SPLINE
SPL {X  -159.063, Y  +688.696, Z    +0.000, E1   +17.094, E3 -430810.553}
SPL {X  -159.987, Y  +672.488, Z    +0.000, E1    +5.638, E3 -430834.618}
SPL {X  -159.990, Y  +663.928, Z    +0.000, E1    -0.338, E3 -430840.413}
SPL {X  -159.990, Y  +658.009, Z    +0.000, E1    -4.774, E3 -430844.113}
SPL {X  -159.990, Y  +651.567, Z    +0.000, E1    -9.674, E3 -430849.516}
SPL {X  -159.990, Y  +638.711, Z    +0.000, E1   -17.883, E3 -430865.162}
SPL {X  -159.990, Y  +631.642, Z    +0.000, E1   -20.884, E3 -430880.721}
SPL {X  -159.990, Y  +626.048, Z    +0.000, E1   -22.026, E3 -430900.714}
SPL {X  -159.990, Y  +623.760, Z    +0.000, E1   -22.031, E3 -430912.701}
SPL {X  -159.990, Y  +621.334, Z    +0.000, E1   -22.029, E3 -430925.427}
SPL {X  -159.990, Y  +618.387, Z    +0.000, E1   -22.057, E3 -430940.817}
SPL {X  -159.990, Y  +615.830, Z    +0.000, E1   -22.023, E3 -430954.309}
SPL {X  -159.990, Y  +614.007, Z    +0.000, E1   -22.018, E3 -430963.886}
SPL {X  -159.990, Y  +611.459, Z    +0.000, E1   -22.053, E3 -430977.173}
SPL {X  -159.990, Y  +608.810, Z    +0.000, E1   -22.023, E3 -430991.141}
SPL {X  -159.990, Y  +606.481, Z    +0.000, E1   -22.033, E3 -431003.316}
SPL {X  -159.990, Y  +603.419, Z    +0.000, E1   -22.064, E3 -431019.256}
SPL {X  -159.990, Y  +600.642, Z    +0.000, E1   -22.032, E3 -431033.885}
SPL {X  -159.990, Y  +598.568, Z    +0.000, E1   -22.046, E3 -431044.678}
SPL {X  -159.990, Y  +595.493, Z    +0.000, E1   -22.070, E3 -431060.761}
SPL {X  -159.990, Y  +592.865, Z    +0.000, E1   -22.036, E3 -431074.590}
SPL {X  -159.990, Y  +590.803, Z    +0.000, E1   -22.046, E3 -431085.381}
SPL {X  -159.990, Y  +587.778, Z    +0.000, E1   -22.073, E3 -431101.156}
SPL {X  -159.990, Y  +585.120, Z    +0.000, E1   -22.045, E3 -431115.100}
SPL {X  -159.990, Y  +583.118, Z    +0.000, E1   -22.052, E3 -431125.586}
SPL {X  -159.990, Y  +580.862, Z    +0.000, E1   -22.049, E3 -431137.424}
SPL {X  -159.990, Y  +578.386, Z    +0.000, E1   -22.057, E3 -431150.379}
SPL {X  -159.990, Y  +576.252, Z    +0.000, E1   -22.038, E3 -431161.602}
SPL {X  -159.990, Y  +574.280, Z    +0.000, E1   -22.051, E3 -431171.896}
SPL {X  -159.990, Y  +571.711, Z    +0.000, E1   -22.058, E3 -431185.370}
SPL {X  -159.990, Y  +569.285, Z    +0.000, E1   -22.044, E3 -431198.095}
SPL {X  -159.990, Y  +567.211, Z    +0.000, E1   -22.046, E3 -431208.956}
SPL {X  -159.990, Y  +565.039, Z    +0.000, E1   -22.047, E3 -431220.334}
SPL {X  -159.990, Y  +562.755, Z    +0.000, E1   -22.047, E3 -431232.319}
SPL {X  -159.990, Y  +560.652, Z    +0.000, E1   -22.038, E3 -431243.364}
SPL {X  -159.990, Y  +558.852, Z    +0.000, E1   -22.046, E3 -431252.736}
SPL {X  -159.990, Y  +556.672, Z    +0.000, E1   -22.055, E3 -431264.126}
SPL {X  -159.990, Y  +553.726, Z    +0.000, E1   -22.080, E3 -431279.488}
SPL {X  -159.990, Y  +550.886, Z    +0.000, E1   -22.056, E3 -431294.427}
SPL {X  -159.990, Y  +547.986, Z    +0.000, E1   -22.078, E3 -431309.546}
SPL {X  -159.990, Y  +545.350, Z    +0.000, E1   -22.053, E3 -431323.407}
SPL {X  -159.990, Y  +543.405, Z    +0.000, E1   -22.048, E3 -431333.620}
SPL {X  -159.990, Y  +541.673, Z    +0.000, E1   -22.053, E3 -431342.684}
SPL {X  -159.990, Y  +539.341, Z    +0.000, E1   -22.056, E3 -431354.889}
SPL {X  -159.990, Y  +536.984, Z    +0.000, E1   -22.057, E3 -431367.221}
SPL {X  -159.990, Y  +534.045, Z    +0.000, E1   -22.087, E3 -431382.545}
SPL {X  -159.990, Y  +530.476, Z    +0.000, E1   -22.084, E3 -431401.239}
SPL {X  -159.990, Y  +527.412, Z    +0.000, E1   -22.067, E3 -431417.302}
SPL {X  -159.990, Y  +524.425, Z    +0.000, E1   -22.078, E3 -431432.935}
SPL {X  -159.990, Y  +521.599, Z    +0.000, E1   -22.060, E3 -431447.777}
SPL {X  -159.990, Y  +519.209, Z    +0.000, E1   -22.063, E3 -431460.252}
SPL {X  -159.990, Y  +516.651, Z    +0.000, E1   -22.071, E3 -431473.631}
SPL {X  -159.990, Y  +514.122, Z    +0.000, E1   -22.061, E3 -431486.903}
SPL {X  -159.990, Y  +511.670, Z    +0.000, E1   -22.064, E3 -431499.753}
SPL {X  -159.990, Y  +506.947, Z    +0.000, E1   -23.726, E3 -431509.781}
SPL {X  -159.990, Y  +496.921, Z    +0.000, E1   -28.340, E3 -431518.530}
SPL {X  -159.990, Y  +495.822, Z    +0.000, E1   -27.449, E3 -431529.278}
SPL {X  -159.990, Y  +494.952, Z    +0.000, E1   -26.628, E3 -431538.861}
SPL {X  -159.990, Y  +493.896, Z    +0.000, E1   -25.736, E3 -431550.191}
SPL {X  -159.990, Y  +491.647, Z    +0.000, E1   -25.401, E3 -431562.726}
SPL {X  -159.990, Y  +488.807, Z    +0.000, E1   -25.397, E3 -431575.425}
SPL {X  -159.990, Y  +486.070, Z    +0.000, E1   -25.399, E3 -431587.656}
SPL {X  -159.990, Y  +483.747, Z    +0.000, E1   -25.384, E3 -431598.069}
SPL {X  -159.990, Y  +481.038, Z    +0.000, E1   -25.412, E3 -431610.124}
SPL {X  -159.990, Y  +477.508, Z    +0.000, E1   -25.410, E3 -431625.906}
SPL {X  -159.990, Y  +473.634, Z    +0.000, E1   -25.426, E3 -431643.195}
SPL {X  -159.990, Y  +470.047, Z    +0.000, E1   -25.402, E3 -431659.276}
SPL {X  -159.990, Y  +467.082, Z    +0.000, E1   -25.399, E3 -431672.523}
SPL {X  -159.990, Y  +464.063, Z    +0.000, E1   -25.405, E3 -431686.018}
SPL {X  -159.990, Y  +460.712, Z    +0.000, E1   -25.411, E3 -431700.978}
SPL {X  -159.990, Y  +457.497, Z    +0.000, E1   -25.403, E3 -431715.350}
SPL {X  -159.990, Y  +455.126, Z    +0.000, E1   -25.389, E3 -431725.959}
SPL {X  -159.990, Y  +452.123, Z    +0.000, E1   -25.426, E3 -431739.317}
SPL {X  -159.990, Y  +448.503, Z    +0.000, E1   -25.410, E3 -431755.518}
SPL {X  -159.990, Y  +445.108, Z    +0.000, E1   -25.407, E3 -431770.756}
SPL {X  -159.990, Y  +441.797, Z    +0.000, E1   -25.390, E3 -431785.635}
SPL {X  -159.990, Y  +439.442, Z    +0.000, E1   -25.369, E3 -431796.212}
SPL {X  -159.990, Y  +436.316, Z    +0.000, E1   -25.420, E3 -431810.094}
SPL {X  -159.990, Y  +432.613, Z    +0.000, E1   -25.390, E3 -431826.719}
SPL {X  -159.990, Y  +429.079, Z    +0.000, E1   -25.407, E3 -431842.490}
SPL {X  -159.990, Y  +425.142, Z    +0.000, E1   -25.407, E3 -431860.092}
SPL {X  -159.990, Y  +421.010, Z    +0.000, E1   -25.418, E3 -431878.554}
SPL {X  -159.990, Y  +417.514, Z    +0.000, E1   -25.386, E3 -431894.246}
SPL {X  -159.990, Y  +414.805, Z    +0.000, E1   -25.385, E3 -431906.367}
SPL {X  -159.990, Y  +411.959, Z    +0.000, E1   -25.386, E3 -431919.093}
SPL {X  -159.990, Y  +408.981, Z    +0.000, E1   -25.392, E3 -431932.397}
SPL {X  -159.990, Y  +405.773, Z    +0.000, E1   -25.398, E3 -431946.707}
SPL {X  -159.990, Y  +402.805, Z    +0.000, E1   -25.389, E3 -431959.993}
SPL {X  -159.990, Y  +400.083, Z    +0.000, E1   -25.388, E3 -431972.170}
SPL {X  -159.990, Y  +396.740, Z    +0.000, E1   -25.410, E3 -431987.094}
SPL {X  -159.990, Y  +392.622, Z    +0.000, E1   -25.413, E3 -432005.522}
SPL {X  -159.990, Y  +388.328, Z    +0.000, E1   -25.413, E3 -432024.750}
SPL {X  -159.990, Y  +384.900, Z    +0.000, E1   -25.383, E3 -432040.112}
SPL {X  -159.990, Y  +382.110, Z    +0.000, E1   -25.393, E3 -432052.559}
SPL {X  -159.961, Y  +379.439, Z    +0.000, E1   -25.380, E3 -432064.538}
SPL {X  -159.894, Y  +376.959, Z    +0.000, E1   -25.370, E3 -432075.715}
SPL {X  -159.784, Y  +374.382, Z    +0.000, E1   -25.356, E3 -432087.356}
SPL {X  -159.621, Y  +371.640, Z    +0.000, E1   -25.335, E3 -432099.796}
SPL {X  -159.406, Y  +368.844, Z    +0.000, E1   -25.307, E3 -432112.509}
SPL {X  -159.144, Y  +366.072, Z    +0.000, E1   -25.281, E3 -432125.117}
SPL {X  -158.822, Y  +363.200, Z    +0.000, E1   -25.236, E3 -432138.289}
SPL {X  -158.491, Y  +360.654, Z    +0.000, E1   -25.188, E3 -432150.029}
SPL {X  -158.127, Y  +358.155, Z    +0.000, E1   -25.126, E3 -432161.649}
SPL {X  -158.095, Y  +357.947, Z    +0.000, E1   -21.741, E3 -432193.221}
ENDSPLINE

SPLINE
SPL {X  -158.454, Y  +360.384, Z    +0.000, E1   -19.366, E3 -432205.372}
SPL {X  -159.737, Y  +373.507, Z    +0.000, E1   -10.311, E3 -432227.408}
SPL {X  -159.990, Y  +382.574, Z    +0.000, E1    -4.463, E3 -432234.095}
SPL {X  -159.990, Y  +387.496, Z    +0.000, E1    -1.004, E3 -432236.841}
SPL {X  -159.990, Y  +395.121, Z    +0.000, E1    +4.514, E3 -432241.153}
SPL {X  -159.990, Y  +407.941, Z    +0.000, E1   +14.126, E3 -432253.227}
SPL {X  -159.990, Y  +418.671, Z    +0.000, E1   +19.855, E3 -432272.643}
SPL {X  -159.990, Y  +429.878, Z    +0.000, E1   +23.330, E3 -432302.698}
SPL {X  -159.990, Y  +432.766, Z    +0.000, E1   +23.321, E3 -432316.921}
SPL {X  -159.990, Y  +435.585, Z    +0.000, E1   +23.327, E3 -432330.801}
SPL {X  -159.990, Y  +439.169, Z    +0.000, E1   +23.353, E3 -432348.383}
SPL {X  -159.990, Y  +442.945, Z    +0.000, E1   +23.339, E3 -432367.001}
SPL {X  -159.990, Y  +446.037, Z    +0.000, E1   +23.324, E3 -432382.251}
SPL {X  -159.990, Y  +448.797, Z    +0.000, E1   +23.331, E3 -432395.781}
SPL {X  -159.990, Y  +451.747, Z    +0.000, E1   +23.333, E3 -432410.329}
SPL {X  -159.990, Y  +455.185, Z    +0.000, E1   +23.350, E3 -432427.189}
SPL {X  -159.990, Y  +458.265, Z    +0.000, E1   +23.328, E3 -432442.376}
SPL {X  -159.990, Y  +460.492, Z    +0.000, E1   +23.317, E3 -432453.375}
SPL {X  -159.990, Y  +462.929, Z    +0.000, E1   +23.331, E3 -432465.331}
SPL {X  -159.990, Y  +466.197, Z    +0.000, E1   +23.351, E3 -432481.368}
SPL {X  -159.990, Y  +468.951, Z    +0.000, E1   +23.319, E3 -432494.986}
SPL {X  -159.990, Y  +470.991, Z    +0.000, E1   +23.322, E3 -432505.015}
SPL {X  -159.990, Y  +474.027, Z    +0.000, E1   +23.352, E3 -432519.919}
SPL {X  -159.990, Y  +477.600, Z    +0.000, E1   +23.351, E3 -432537.523}
SPL {X  -159.990, Y  +481.169, Z    +0.000, E1   +23.337, E3 -432555.120}
SPL {X  -159.990, Y  +483.782, Z    +0.000, E1   +23.316, E3 -432568.025}
SPL {X  -159.990, Y  +486.109, Z    +0.000, E1   +23.322, E3 -432579.477}
SPL {X  -159.990, Y  +489.247, Z    +0.000, E1   +23.348, E3 -432594.864}
SPL {X  -159.990, Y  +493.031, Z    +0.000, E1   +23.350, E3 -432613.488}
SPL {X  -159.990, Y  +496.869, Z    +0.000, E1   +23.349, E3 -432632.379}
SPL {X  -159.990, Y  +499.995, Z    +0.000, E1   +23.324, E3 -432647.812}
SPL {X  -159.990, Y  +502.456, Z    +0.000, E1   +23.324, E3 -432659.927}
SPL {X  -159.990, Y  +504.508, Z    +0.000, E1   +23.311, E3 -432670.061}
SPL {X  -159.990, Y  +506.420, Z    +0.000, E1   +23.317, E3 -432679.453}
SPL {X  -159.990, Y  +508.862, Z    +0.000, E1   +23.328, E3 -432691.446}
SPL {X  -159.990, Y  +511.771, Z    +0.000, E1   +23.331, E3 -432705.768}
SPL {X  -159.990, Y  +514.757, Z    +0.000, E1   +23.329, E3 -432720.476}
SPL {X  -159.990, Y  +517.536, Z    +0.000, E1   +23.326, E3 -432734.142}
SPL {X  -159.990, Y  +519.961, Z    +0.000, E1   +23.334, E3 -432745.995}
SPL {X  -159.990, Y  +521.849, Z    +0.000, E1   +23.320, E3 -432755.317}
SPL {X  -159.990, Y  +523.968, Z    +0.000, E1   +23.332, E3 -432765.753}
SPL {X  -159.990, Y  +526.466, Z    +0.000, E1   +23.320, E3 -432778.096}
SPL {X  -159.990, Y  +528.815, Z    +0.000, E1   +23.322, E3 -432789.656}
SPL {X  -159.990, Y  +531.246, Z    +0.000, E1   +23.325, E3 -432801.594}
SPL {X  -159.990, Y  +534.143, Z    +0.000, E1   +23.341, E3 -432815.829}
SPL {X  -159.990, Y  +537.024, Z    +0.000, E1   +23.321, E3 -432830.073}
SPL {X  -159.990, Y  +539.129, Z    +0.000, E1   +23.310, E3 -432840.456}
SPL {X  -159.990, Y  +541.183, Z    +0.000, E1   +23.319, E3 -432850.553}
SPL {X  -159.990, Y  +544.314, Z    +0.000, E1   +23.352, E3 -432865.881}
SPL {X  -159.990, Y  +548.126, Z    +0.000, E1   +23.354, E3 -432884.636}
SPL {X  -159.990, Y  +551.344, Z    +0.000, E1   +23.327, E3 -432900.528}
SPL {X  -159.990, Y  +553.642, Z    +0.000, E1   +23.319, E3 -432911.847}
SPL {X  -159.990, Y  +556.481, Z    +0.000, E1   +23.354, E3 -432925.754}
SPL {X  -159.990, Y  +559.475, Z    +0.000, E1   +23.321, E3 -432940.559}
SPL {X  -159.990, Y  +561.830, Z    +0.000, E1   +23.325, E3 -432952.144}
SPL {X  -159.990, Y  +564.273, Z    +0.000, E1   +23.325, E3 -432964.168}
SPL {X  -159.990, Y  +567.351, Z    +0.000, E1   +23.348, E3 -432979.264}
SPL {X  -159.990, Y  +570.560, Z    +0.000, E1   +23.333, E3 -432995.093}
SPL {X  -159.990, Y  +572.975, Z    +0.000, E1   +23.316, E3 -433007.013}
SPL {X  -159.990, Y  +575.097, Z    +0.000, E1   +23.325, E3 -433017.440}
SPL {X  -159.990, Y  +577.540, Z    +0.000, E1   +23.325, E3 -433029.468}
SPL {X  -159.990, Y  +580.312, Z    +0.000, E1   +23.340, E3 -433043.050}
SPL {X  -159.990, Y  +583.018, Z    +0.000, E1   +23.331, E3 -433056.355}
SPL {X  -159.990, Y  +585.165, Z    +0.000, E1   +23.322, E3 -433066.971}
SPL {X  -159.990, Y  +587.388, Z    +0.000, E1   +23.328, E3 -433077.883}
SPL {X  -159.990, Y  +589.763, Z    +0.000, E1   +23.328, E3 -433089.570}
SPL {X  -159.990, Y  +592.397, Z    +0.000, E1   +23.344, E3 -433102.451}
SPL {X  -159.990, Y  +595.589, Z    +0.000, E1   +23.356, E3 -433118.124}
SPL {X  -159.990, Y  +598.571, Z    +0.000, E1   +23.347, E3 -433132.767}
SPL {X  -159.990, Y  +600.935, Z    +0.000, E1   +23.343, E3 -433144.360}
SPL {X  -159.990, Y  +603.047, Z    +0.000, E1   +23.344, E3 -433154.746}
SPL {X  -159.990, Y  +605.187, Z    +0.000, E1   +23.344, E3 -433165.268}
SPL {X  -159.990, Y  +607.319, Z    +0.000, E1   +23.353, E3 -433175.730}
SPL {X  -159.990, Y  +609.514, Z    +0.000, E1   +23.337, E3 -433186.560}
SPL {X  -159.990, Y  +611.376, Z    +0.000, E1   +23.336, E3 -433195.747}
SPL {X  -159.990, Y  +613.591, Z    +0.000, E1   +23.342, E3 -433206.624}
SPL {X  -159.990, Y  +615.604, Z    +0.000, E1   +23.330, E3 -433216.562}
SPL {X  -159.990, Y  +617.623, Z    +0.000, E1   +23.337, E3 -433226.492}
SPL {X  -159.990, Y  +620.788, Z    +0.000, E1   +23.368, E3 -433241.997}
SPL {X  -159.990, Y  +623.764, Z    +0.000, E1   +23.335, E3 -433256.690}
SPL {X  -159.990, Y  +625.941, Z    +0.000, E1   +23.337, E3 -433267.381}
SPL {X  -159.990, Y  +628.611, Z    +0.000, E1   +23.357, E3 -433280.460}
SPL {X  -159.990, Y  +631.169, Z    +0.000, E1   +23.338, E3 -433293.064}
SPL {X  -159.990, Y  +633.318, Z    +0.000, E1   +23.339, E3 -433303.653}
SPL {X  -159.990, Y  +635.650, Z    +0.000, E1   +23.339, E3 -433315.124}
SPL {X  -159.990, Y  +637.839, Z    +0.000, E1   +23.335, E3 -433325.934}
SPL {X  -159.990, Y  +640.072, Z    +0.000, E1   +23.325, E3 -433336.966}
SPL {X  -159.990, Y  +642.230, Z    +0.000, E1   +23.323, E3 -433347.648}
SPL {X  -159.990, Y  +645.287, Z    +0.000, E1   +23.340, E3 -433362.674}
SPL {X  -159.990, Y  +648.792, Z    +0.000, E1   +23.346, E3 -433379.933}
SPL {X  -159.990, Y  +652.623, Z    +0.000, E1   +23.348, E3 -433398.768}
SPL {X  -159.990, Y  +656.380, Z    +0.000, E1   +23.347, E3 -433417.262}
SPL {X  -159.990, Y  +659.180, Z    +0.000, E1   +23.314, E3 -433431.110}
SPL {X  -159.990, Y  +661.392, Z    +0.000, E1   +23.318, E3 -433442.004}
SPL {X  -159.990, Y  +663.662, Z    +0.000, E1   +23.322, E3 -433453.128}
SPL {X  -159.990, Y  +665.964, Z    +0.000, E1   +23.328, E3 -433464.419}
SPL {X  -159.990, Y  +668.989, Z    +0.000, E1   +23.359, E3 -433479.254}
SPL {X  -159.990, Y  +671.893, Z    +0.000, E1   +23.319, E3 -433493.634}
SPL {X  -159.974, Y  +673.789, Z    +0.000, E1   +23.323, E3 -433502.950}
SPL {X  -159.924, Y  +676.110, Z    +0.000, E1   +23.320, E3 -433514.435}
SPL {X  -159.801, Y  +679.265, Z    +0.000, E1   +23.327, E3 -433530.053}
SPL {X  -159.626, Y  +682.287, Z    +0.000, E1   +23.280, E3 -433545.152}
SPL {X  -159.462, Y  +684.486, Z    +0.000, E1   +23.258, E3 -433556.152}
SPL {X  -159.246, Y  +686.911, Z    +0.000, E1   +23.230, E3 -433568.313}
SPL {X  -159.019, Y  +689.098, Z    +0.000, E1   +23.200, E3 -433579.315}
SPL {X  -158.771, Y  +691.210, Z    +0.000, E1   +23.159, E3 -433589.990}
SPL {X  -158.553, Y  +692.896, Z    +0.000, E1   +23.130, E3 -433598.519}
ENDSPLINE

SPLINE
SPL {X  -159.063, Y  +688.696, Z    +0.000, E1   +17.094, E3 -433636.640}
SPL {X  -159.987, Y  +672.488, Z    +0.000, E1    +5.638, E3 -433660.705}
SPL {X  -159.990, Y  +663.928, Z    +0.000, E1    -0.338, E3 -433666.500}
SPL {X  -159.990, Y  +658.009, Z    +0.000, E1    -4.774, E3 -433670.200}
SPL {X  -159.990, Y  +651.567, Z    +0.000, E1    -9.674, E3 -433675.603}
SPL {X  -159.990, Y  +638.711, Z    +0.000, E1   -17.883, E3 -433691.249}
SPL {X  -159.990, Y  +631.642, Z    +0.000, E1   -20.884, E3 -433706.808}
SPL {X  -159.990, Y  +626.048, Z    +0.000, E1   -22.026, E3 -433726.801}
SPL {X  -159.990, Y  +623.760, Z    +0.000, E1   -22.031, E3 -433738.788}
SPL {X  -159.990, Y  +621.334, Z    +0.000, E1   -22.029, E3 -433751.514}
SPL {X  -159.990, Y  +619.505, Z    +0.000, E1   -22.018, E3 -433761.130}
SPL {X  -159.990, Y  +617.621, Z    +0.000, E1   -22.025, E3 -433770.996}
SPL {X  -159.990, Y  +615.830, Z    +0.000, E1   -22.023, E3 -433780.396}
SPL {X  -159.990, Y  +613.034, Z    +0.000, E1   -22.053, E3 -433795.002}
SPL {X  -159.990, Y  +609.503, Z    +0.000, E1   -22.054, E3 -433813.529}
SPL {X  -159.990, Y  +605.804, Z    +0.000, E1   -22.064, E3 -433832.873}
SPL {X  -159.990, Y  +602.819, Z    +0.000, E1   -22.037, E3 -433848.544}
SPL {X  -159.990, Y  +600.642, Z    +0.000, E1   -22.032, E3 -433859.972}
SPL {X  -159.990, Y  +598.568, Z    +0.000, E1   -22.046, E3 -433870.765}
SPL {X  -159.990, Y  +596.440, Z    +0.000, E1   -22.036, E3 -433881.947}
SPL {X  -159.990, Y  +593.768, Z    +0.000, E1   -22.071, E3 -433895.880}
SPL {X  -159.990, Y  +590.068, Z    +0.000, E1   -22.076, E3 -433915.248}
SPL {X  -159.990, Y  +587.130, Z    +0.000, E1   -22.046, E3 -433930.685}
SPL {X  -159.990, Y  +585.120, Z    +0.000, E1   -22.045, E3 -433941.187}
SPL {X  -159.990, Y  +583.118, Z    +0.000, E1   -22.052, E3 -433951.673}
SPL {X  -159.990, Y  +580.862, Z    +0.000, E1   -22.049, E3 -433963.511}
SPL {X  -159.990, Y  +578.386, Z    +0.000, E1   -22.057, E3 -433976.466}
SPL {X  -159.990, Y  +576.252, Z    +0.000, E1   -22.038, E3 -433987.689}
SPL {X  -159.990, Y  +574.280, Z    +0.000, E1   -22.051, E3 -433997.983}
SPL {X  -159.990, Y  +571.711, Z    +0.000, E1   -22.058, E3 -434011.457}
SPL {X  -159.990, Y  +569.285, Z    +0.000, E1   -22.044, E3 -434024.182}
SPL {X  -159.990, Y  +567.211, Z    +0.000, E1   -22.046, E3 -434035.043}
SPL {X  -159.990, Y  +565.039, Z    +0.000, E1   -22.047, E3 -434046.421}
SPL {X  -159.990, Y  +562.755, Z    +0.000, E1   -22.047, E3 -434058.406}
SPL {X  -159.990, Y  +559.661, Z    +0.000, E1   -22.078, E3 -434074.538}
SPL {X  -159.990, Y  +555.965, Z    +0.000, E1   -22.085, E3 -434093.847}
SPL {X  -159.990, Y  +553.115, Z    +0.000, E1   -22.054, E3 -434108.832}
SPL {X  -159.990, Y  +550.886, Z    +0.000, E1   -22.056, E3 -434120.514}
SPL {X  -159.990, Y  +547.986, Z    +0.000, E1   -22.078, E3 -434135.633}
SPL {X  -159.990, Y  +545.350, Z    +0.000, E1   -22.053, E3 -434149.494}
SPL {X  -159.990, Y  +543.405, Z    +0.000, E1   -22.048, E3 -434159.707}
SPL {X  -159.990, Y  +541.673, Z    +0.000, E1   -22.053, E3 -434168.771}
SPL {X  -159.990, Y  +539.341, Z    +0.000, E1   -22.056, E3 -434180.976}
SPL {X  -159.990, Y  +536.301, Z    +0.000, E1   -22.084, E3 -434196.831}
SPL {X  -159.990, Y  +533.389, Z    +0.000, E1   -22.057, E3 -434212.138}
SPL {X  -159.990, Y  +531.347, Z    +0.000, E1   -22.052, E3 -434222.839}
SPL {X  -159.990, Y  +528.972, Z    +0.000, E1   -22.072, E3 -434235.212}
SPL {X  -159.990, Y  +526.034, Z    +0.000, E1   -22.073, E3 -434250.591}
SPL {X  -159.990, Y  +523.717, Z    +0.000, E1   -22.050, E3 -434262.796}
SPL {X  -159.990, Y  +521.599, Z    +0.000, E1   -22.060, E3 -434273.864}
SPL {X  -159.990, Y  +519.209, Z    +0.000, E1   -22.063, E3 -434286.338}
SPL {X  -159.990, Y  +517.330, Z    +0.000, E1   -22.053, E3 -434296.194}
SPL {X  -159.990, Y  +514.729, Z    +0.000, E1   -22.089, E3 -434309.752}
SPL {X  -159.990, Y  +511.670, Z    +0.000, E1   -22.064, E3 -434325.840}
SPL {X  -159.990, Y  +506.947, Z    +0.000, E1   -23.726, E3 -434335.868}
SPL {X  -159.990, Y  +496.921, Z    +0.000, E1   -28.340, E3 -434344.617}
SPL {X  -159.990, Y  +495.822, Z    +0.000, E1   -27.449, E3 -434355.365}
SPL {X  -159.990, Y  +494.952, Z    +0.000, E1   -26.628, E3 -434364.948}
SPL {X  -159.990, Y  +493.896, Z    +0.000, E1   -25.736, E3 -434376.278}
SPL {X  -159.990, Y  +491.647, Z    +0.000, E1   -25.401, E3 -434388.813}
SPL {X  -159.990, Y  +488.807, Z    +0.000, E1   -25.397, E3 -434401.512}
SPL {X  -159.990, Y  +486.070, Z    +0.000, E1   -25.399, E3 -434413.743}
SPL {X  -159.990, Y  +482.821, Z    +0.000, E1   -25.411, E3 -434428.244}
SPL {X  -159.990, Y  +480.183, Z    +0.000, E1   -25.384, E3 -434440.084}
SPL {X  -159.990, Y  +477.508, Z    +0.000, E1   -25.410, E3 -434451.993}
SPL {X  -159.990, Y  +473.634, Z    +0.000, E1   -25.426, E3 -434469.282}
SPL {X  -159.990, Y  +470.047, Z    +0.000, E1   -25.402, E3 -434485.363}
SPL {X  -159.990, Y  +467.082, Z    +0.000, E1   -25.399, E3 -434498.610}
SPL {X  -159.990, Y  +464.063, Z    +0.000, E1   -25.405, E3 -434512.105}
SPL {X  -159.990, Y  +460.712, Z    +0.000, E1   -25.411, E3 -434527.065}
SPL {X  -159.990, Y  +457.497, Z    +0.000, E1   -25.403, E3 -434541.437}
SPL {X  -159.990, Y  +455.126, Z    +0.000, E1   -25.389, E3 -434552.046}
SPL {X  -159.990, Y  +453.438, Z    +0.000, E1   -25.385, E3 -434559.606}
SPL {X  -159.990, Y  +450.823, Z    +0.000, E1   -25.417, E3 -434571.225}
SPL {X  -159.990, Y  +446.894, Z    +0.000, E1   -25.428, E3 -434588.782}
SPL {X  -159.990, Y  +443.345, Z    +0.000, E1   -25.390, E3 -434604.790}
SPL {X  -159.990, Y  +441.077, Z    +0.000, E1   -25.369, E3 -434614.988}
SPL {X  -159.990, Y  +438.608, Z    +0.000, E1   -25.392, E3 -434625.985}
SPL {X  -159.990, Y  +434.852, Z    +0.000, E1   -25.415, E3 -434642.739}
SPL {X  -159.990, Y  +430.645, Z    +0.000, E1   -25.414, E3 -434661.559}
SPL {X  -159.990, Y  +426.865, Z    +0.000, E1   -25.398, E3 -434678.488}
SPL {X  -159.990, Y  +424.251, Z    +0.000, E1   -25.375, E3 -434690.225}
SPL {X  -159.990, Y  +421.010, Z    +0.000, E1   -25.418, E3 -434704.640}
SPL {X  -159.990, Y  +417.514, Z    +0.000, E1   -25.386, E3 -434720.333}
SPL {X  -159.990, Y  +414.805, Z    +0.000, E1   -25.385, E3 -434732.453}
SPL {X  -159.990, Y  +411.282, Z    +0.000, E1   -25.413, E3 -434748.154}
SPL {X  -159.990, Y  +408.351, Z    +0.000, E1   -25.372, E3 -434761.341}
SPL {X  -159.990, Y  +405.773, Z    +0.000, E1   -25.398, E3 -434772.794}
SPL {X  -159.990, Y  +402.805, Z    +0.000, E1   -25.389, E3 -434786.080}
SPL {X  -159.990, Y  +400.083, Z    +0.000, E1   -25.388, E3 -434798.257}
SPL {X  -159.990, Y  +396.740, Z    +0.000, E1   -25.410, E3 -434813.181}
SPL {X  -159.990, Y  +393.569, Z    +0.000, E1   -25.379, E3 -434827.431}
SPL {X  -159.990, Y  +390.564, Z    +0.000, E1   -25.393, E3 -434840.875}
SPL {X  -159.990, Y  +387.503, Z    +0.000, E1   -25.378, E3 -434854.589}
SPL {X  -159.990, Y  +384.900, Z    +0.000, E1   -25.383, E3 -434866.199}
SPL {X  -159.990, Y  +382.110, Z    +0.000, E1   -25.393, E3 -434878.646}
SPL {X  -159.961, Y  +379.439, Z    +0.000, E1   -25.380, E3 -434890.625}
SPL {X  -159.894, Y  +376.959, Z    +0.000, E1   -25.370, E3 -434901.802}
SPL {X  -159.784, Y  +374.382, Z    +0.000, E1   -25.356, E3 -434913.443}
SPL {X  -159.621, Y  +371.640, Z    +0.000, E1   -25.335, E3 -434925.883}
SPL {X  -159.406, Y  +368.844, Z    +0.000, E1   -25.307, E3 -434938.596}
SPL {X  -159.144, Y  +366.072, Z    +0.000, E1   -25.281, E3 -434951.204}
SPL {X  -158.822, Y  +363.200, Z    +0.000, E1   -25.236, E3 -434964.376}
SPL {X  -158.491, Y  +360.654, Z    +0.000, E1   -25.188, E3 -434976.116}
SPL {X  -158.127, Y  +358.155, Z    +0.000, E1   -25.126, E3 -434987.736}
SPL {X  -158.095, Y  +357.947, Z    +0.000, E1   -21.741, E3 -435019.308}
ENDSPLINE

SPLINE
SPL {X  -158.454, Y  +360.384, Z    +0.000, E1   -19.366, E3 -435031.459}
SPL {X  -159.737, Y  +373.507, Z    +0.000, E1   -10.311, E3 -435053.495}
SPL {X  -159.990, Y  +382.574, Z    +0.000, E1    -4.463, E3 -435060.182}
SPL {X  -159.990, Y  +389.909, Z    +0.000, E1    +0.662, E3 -435064.197}
SPL {X  -159.990, Y  +396.289, Z    +0.000, E1    +5.500, E3 -435067.977}
SPL {X  -159.990, Y  +407.941, Z    +0.000, E1   +14.126, E3 -435079.314}
SPL {X  -159.990, Y  +418.671, Z    +0.000, E1   +19.855, E3 -435098.730}
SPL {X  -159.990, Y  +429.878, Z    +0.000, E1   +23.330, E3 -435128.785}
SPL {X  -159.990, Y  +432.103, Z    +0.000, E1   +23.301, E3 -435139.804}
SPL {X  -159.990, Y  +434.188, Z    +0.000, E1   +23.325, E3 -435150.000}
SPL {X  -159.990, Y  +436.320, Z    +0.000, E1   +23.304, E3 -435160.553}
SPL {X  -159.990, Y  +439.169, Z    +0.000, E1   +23.353, E3 -435174.470}
SPL {X  -159.990, Y  +442.945, Z    +0.000, E1   +23.339, E3 -435193.088}
SPL {X  -159.990, Y  +446.037, Z    +0.000, E1   +23.324, E3 -435208.338}
SPL {X  -159.990, Y  +448.797, Z    +0.000, E1   +23.331, E3 -435221.868}
SPL {X  -159.990, Y  +451.747, Z    +0.000, E1   +23.333, E3 -435236.416}
SPL {X  -159.990, Y  +455.185, Z    +0.000, E1   +23.350, E3 -435253.276}
SPL {X  -159.990, Y  +458.265, Z    +0.000, E1   +23.328, E3 -435268.463}
SPL {X  -159.990, Y  +460.492, Z    +0.000, E1   +23.317, E3 -435279.462}
SPL {X  -159.990, Y  +462.929, Z    +0.000, E1   +23.331, E3 -435291.418}
SPL {X  -159.990, Y  +465.027, Z    +0.000, E1   +23.313, E3 -435301.771}
SPL {X  -159.990, Y  +466.881, Z    +0.000, E1   +23.322, E3 -435310.880}
SPL {X  -159.990, Y  +468.951, Z    +0.000, E1   +23.319, E3 -435321.072}
SPL {X  -159.990, Y  +471.818, Z    +0.000, E1   +23.351, E3 -435335.119}
SPL {X  -159.990, Y  +474.801, Z    +0.000, E1   +23.320, E3 -435349.895}
SPL {X  -159.990, Y  +476.830, Z    +0.000, E1   +23.323, E3 -435359.874}
SPL {X  -159.990, Y  +479.553, Z    +0.000, E1   +23.328, E3 -435373.276}
SPL {X  -159.990, Y  +481.893, Z    +0.000, E1   +23.312, E3 -435384.826}
SPL {X  -159.990, Y  +483.782, Z    +0.000, E1   +23.316, E3 -435394.112}
SPL {X  -159.990, Y  +486.109, Z    +0.000, E1   +23.322, E3 -435405.564}
SPL {X  -159.990, Y  +489.247, Z    +0.000, E1   +23.348, E3 -435420.951}
SPL {X  -159.990, Y  +493.031, Z    +0.000, E1   +23.350, E3 -435439.575}
SPL {X  -159.990, Y  +496.869, Z    +0.000, E1   +23.349, E3 -435458.466}
SPL {X  -159.990, Y  +499.995, Z    +0.000, E1   +23.324, E3 -435473.899}
SPL {X  -159.990, Y  +502.456, Z    +0.000, E1   +23.324, E3 -435486.014}
SPL {X  -159.990, Y  +505.646, Z    +0.000, E1   +23.350, E3 -435501.669}
SPL {X  -159.990, Y  +508.862, Z    +0.000, E1   +23.328, E3 -435517.533}
SPL {X  -159.990, Y  +511.771, Z    +0.000, E1   +23.331, E3 -435531.855}
SPL {X  -159.990, Y  +514.016, Z    +0.000, E1   +23.308, E3 -435542.959}
SPL {X  -159.990, Y  +516.860, Z    +0.000, E1   +23.355, E3 -435556.845}
SPL {X  -159.990, Y  +520.719, Z    +0.000, E1   +23.363, E3 -435575.755}
SPL {X  -159.990, Y  +523.968, Z    +0.000, E1   +23.332, E3 -435591.840}
SPL {X  -159.990, Y  +526.466, Z    +0.000, E1   +23.320, E3 -435604.183}
SPL {X  -159.990, Y  +528.815, Z    +0.000, E1   +23.322, E3 -435615.743}
SPL {X  -159.990, Y  +531.246, Z    +0.000, E1   +23.325, E3 -435627.681}
SPL {X  -159.990, Y  +533.354, Z    +0.000, E1   +23.318, E3 -435638.067}
SPL {X  -159.990, Y  +534.931, Z    +0.000, E1   +23.312, E3 -435645.861}
SPL {X  -159.990, Y  +537.024, Z    +0.000, E1   +23.321, E3 -435656.160}
SPL {X  -159.990, Y  +539.129, Z    +0.000, E1   +23.310, E3 -435666.543}
SPL {X  -159.990, Y  +541.183, Z    +0.000, E1   +23.319, E3 -435676.640}
SPL {X  -159.990, Y  +544.314, Z    +0.000, E1   +23.352, E3 -435691.968}
SPL {X  -159.990, Y  +548.126, Z    +0.000, E1   +23.354, E3 -435710.723}
SPL {X  -159.990, Y  +551.344, Z    +0.000, E1   +23.327, E3 -435726.615}
SPL {X  -159.990, Y  +553.642, Z    +0.000, E1   +23.319, E3 -435737.934}
SPL {X  -159.990, Y  +556.481, Z    +0.000, E1   +23.354, E3 -435751.841}
SPL {X  -159.990, Y  +559.475, Z    +0.000, E1   +23.321, E3 -435766.646}
SPL {X  -159.990, Y  +561.830, Z    +0.000, E1   +23.325, E3 -435778.231}
SPL {X  -159.990, Y  +564.273, Z    +0.000, E1   +23.325, E3 -435790.255}
SPL {X  -159.990, Y  +567.351, Z    +0.000, E1   +23.348, E3 -435805.351}
SPL {X  -159.990, Y  +570.560, Z    +0.000, E1   +23.333, E3 -435821.180}
SPL {X  -159.990, Y  +572.975, Z    +0.000, E1   +23.316, E3 -435833.100}
SPL {X  -159.990, Y  +575.097, Z    +0.000, E1   +23.325, E3 -435843.527}
SPL {X  -159.990, Y  +577.540, Z    +0.000, E1   +23.325, E3 -435855.555}
SPL {X  -159.990, Y  +580.312, Z    +0.000, E1   +23.340, E3 -435869.137}
SPL {X  -159.990, Y  +583.018, Z    +0.000, E1   +23.331, E3 -435882.442}
SPL {X  -159.990, Y  +585.165, Z    +0.000, E1   +23.322, E3 -435893.058}
SPL {X  -159.990, Y  +587.388, Z    +0.000, E1   +23.328, E3 -435903.970}
SPL {X  -159.990, Y  +589.763, Z    +0.000, E1   +23.328, E3 -435915.657}
SPL {X  -159.990, Y  +592.397, Z    +0.000, E1   +23.344, E3 -435928.538}
SPL {X  -159.990, Y  +595.589, Z    +0.000, E1   +23.356, E3 -435944.211}
SPL {X  -159.990, Y  +598.571, Z    +0.000, E1   +23.347, E3 -435958.854}
SPL {X  -159.990, Y  +600.935, Z    +0.000, E1   +23.343, E3 -435970.447}
SPL {X  -159.990, Y  +603.047, Z    +0.000, E1   +23.344, E3 -435980.833}
SPL {X  -159.990, Y  +605.187, Z    +0.000, E1   +23.344, E3 -435991.355}
SPL {X  -159.990, Y  +607.319, Z    +0.000, E1   +23.353, E3 -436001.817}
SPL {X  -159.990, Y  +609.514, Z    +0.000, E1   +23.337, E3 -436012.646}
SPL {X  -159.990, Y  +611.376, Z    +0.000, E1   +23.336, E3 -436021.834}
SPL {X  -159.990, Y  +613.591, Z    +0.000, E1   +23.342, E3 -436032.711}
SPL {X  -159.990, Y  +615.604, Z    +0.000, E1   +23.330, E3 -436042.649}
SPL {X  -159.990, Y  +617.623, Z    +0.000, E1   +23.337, E3 -436052.579}
SPL {X  -159.990, Y  +620.788, Z    +0.000, E1   +23.368, E3 -436068.084}
SPL {X  -159.990, Y  +623.764, Z    +0.000, E1   +23.335, E3 -436082.777}
SPL {X  -159.990, Y  +625.941, Z    +0.000, E1   +23.337, E3 -436093.468}
SPL {X  -159.990, Y  +628.611, Z    +0.000, E1   +23.357, E3 -436106.547}
SPL {X  -159.990, Y  +631.169, Z    +0.000, E1   +23.338, E3 -436119.151}
SPL {X  -159.990, Y  +633.318, Z    +0.000, E1   +23.339, E3 -436129.740}
SPL {X  -159.990, Y  +635.650, Z    +0.000, E1   +23.339, E3 -436141.211}
SPL {X  -159.990, Y  +637.839, Z    +0.000, E1   +23.335, E3 -436152.021}
SPL {X  -159.990, Y  +640.072, Z    +0.000, E1   +23.325, E3 -436163.053}
SPL {X  -159.990, Y  +642.230, Z    +0.000, E1   +23.323, E3 -436173.735}
SPL {X  -159.990, Y  +645.287, Z    +0.000, E1   +23.340, E3 -436188.761}
SPL {X  -159.990, Y  +648.792, Z    +0.000, E1   +23.346, E3 -436206.020}
SPL {X  -159.990, Y  +652.623, Z    +0.000, E1   +23.348, E3 -436224.854}
SPL {X  -159.990, Y  +656.380, Z    +0.000, E1   +23.347, E3 -436243.349}
SPL {X  -159.990, Y  +659.180, Z    +0.000, E1   +23.314, E3 -436257.197}
SPL {X  -159.990, Y  +661.392, Z    +0.000, E1   +23.318, E3 -436268.091}
SPL {X  -159.990, Y  +663.662, Z    +0.000, E1   +23.322, E3 -436279.215}
SPL {X  -159.990, Y  +665.964, Z    +0.000, E1   +23.328, E3 -436290.506}
SPL {X  -159.990, Y  +668.989, Z    +0.000, E1   +23.359, E3 -436305.341}
SPL {X  -159.983, Y  +672.946, Z    +0.000, E1   +23.359, E3 -436324.823}
SPL {X  -159.924, Y  +676.110, Z    +0.000, E1   +23.320, E3 -436340.522}
SPL {X  -159.801, Y  +679.265, Z    +0.000, E1   +23.327, E3 -436356.140}
SPL {X  -159.626, Y  +682.287, Z    +0.000, E1   +23.280, E3 -436371.239}
SPL {X  -159.462, Y  +684.486, Z    +0.000, E1   +23.258, E3 -436382.239}
SPL {X  -159.246, Y  +686.911, Z    +0.000, E1   +23.230, E3 -436394.400}
SPL {X  -159.019, Y  +689.098, Z    +0.000, E1   +23.200, E3 -436405.402}
SPL {X  -158.660, Y  +692.086, Z    +0.000, E1   +23.176, E3 -436420.446}
ENDSPLINE

SPLINE
SPL {X  -159.063, Y  +688.696, Z    +0.000, E1   +17.094, E3 -436462.727}
SPL {X  -159.967, Y  +674.206, Z    +0.000, E1    +6.731, E3 -436485.540}
SPL {X  -159.990, Y  +665.270, Z    +0.000, E1    +0.699, E3 -436491.710}
SPL {X  -159.990, Y  +658.009, Z    +0.000, E1    -4.774, E3 -436496.287}
SPL {X  -159.990, Y  +651.567, Z    +0.000, E1    -9.674, E3 -436501.690}
SPL {X  -159.990, Y  +637.762, Z    +0.000, E1   -18.345, E3 -436519.048}
SPL {X  -159.990, Y  +626.382, Z    +0.000, E1   -22.040, E3 -436551.097}
SPL {X  -159.990, Y  +623.760, Z    +0.000, E1   -22.031, E3 -436564.875}
SPL {X  -159.990, Y  +621.334, Z    +0.000, E1   -22.029, E3 -436577.601}
SPL {X  -159.990, Y  +619.505, Z    +0.000, E1   -22.018, E3 -436587.217}
SPL {X  -159.990, Y  +617.621, Z    +0.000, E1   -22.025, E3 -436597.083}
SPL {X  -159.990, Y  +614.928, Z    +0.000, E1   -22.055, E3 -436611.144}
SPL {X  -159.990, Y  +611.459, Z    +0.000, E1   -22.053, E3 -436629.347}
SPL {X  -159.990, Y  +608.810, Z    +0.000, E1   -22.023, E3 -436643.315}
SPL {X  -159.990, Y  +605.804, Z    +0.000, E1   -22.064, E3 -436658.960}
SPL {X  -159.990, Y  +602.819, Z    +0.000, E1   -22.037, E3 -436674.631}
SPL {X  -159.990, Y  +600.642, Z    +0.000, E1   -22.032, E3 -436686.059}
SPL {X  -159.990, Y  +598.568, Z    +0.000, E1   -22.046, E3 -436696.852}
SPL {X  -159.990, Y  +596.440, Z    +0.000, E1   -22.036, E3 -436708.034}
SPL {X  -159.990, Y  +593.768, Z    +0.000, E1   -22.071, E3 -436721.967}
SPL {X  -159.990, Y  +590.068, Z    +0.000, E1   -22.076, E3 -436741.335}
SPL {X  -159.990, Y  +587.130, Z    +0.000, E1   -22.046, E3 -436756.772}
SPL {X  -159.990, Y  +585.120, Z    +0.000, E1   -22.045, E3 -436767.274}
SPL {X  -159.990, Y  +583.118, Z    +0.000, E1   -22.052, E3 -436777.760}
SPL {X  -159.990, Y  +580.862, Z    +0.000, E1   -22.049, E3 -436789.598}
SPL {X  -159.990, Y  +578.386, Z    +0.000, E1   -22.057, E3 -436802.553}
SPL {X  -159.990, Y  +576.252, Z    +0.000, E1   -22.038, E3 -436813.776}
SPL {X  -159.990, Y  +574.280, Z    +0.000, E1   -22.051, E3 -436824.070}
SPL {X  -159.990, Y  +571.711, Z    +0.000, E1   -22.058, E3 -436837.544}
SPL {X  -159.990, Y  +569.285, Z    +0.000, E1   -22.044, E3 -436850.269}
SPL {X  -159.990, Y  +567.211, Z    +0.000, E1   -22.046, E3 -436861.130}
SPL {X  -159.990, Y  +565.039, Z    +0.000, E1   -22.047, E3 -436872.508}
SPL {X  -159.990, Y  +562.755, Z    +0.000, E1   -22.047, E3 -436884.493}
SPL {X  -159.990, Y  +560.652, Z    +0.000, E1   -22.038, E3 -436895.538}
SPL {X  -159.990, Y  +558.852, Z    +0.000, E1   -22.046, E3 -436904.910}
SPL {X  -159.990, Y  +556.672, Z    +0.000, E1   -22.055, E3 -436916.300}
SPL {X  -159.990, Y  +553.726, Z    +0.000, E1   -22.080, E3 -436931.662}
SPL {X  -159.990, Y  +550.886, Z    +0.000, E1   -22.056, E3 -436946.601}
SPL {X  -159.990, Y  +548.814, Z    +0.000, E1   -22.049, E3 -436957.447}
SPL {X  -159.990, Y  +546.122, Z    +0.000, E1   -22.088, E3 -436971.460}
SPL {X  -159.990, Y  +542.390, Z    +0.000, E1   -22.086, E3 -436991.042}
SPL {X  -159.990, Y  +539.341, Z    +0.000, E1   -22.056, E3 -437007.063}
SPL {X  -159.990, Y  +536.984, Z    +0.000, E1   -22.057, E3 -437019.395}
SPL {X  -159.990, Y  +534.045, Z    +0.000, E1   -22.087, E3 -437034.719}
SPL {X  -159.990, Y  +530.476, Z    +0.000, E1   -22.084, E3 -437053.412}
SPL {X  -159.990, Y  +527.412, Z    +0.000, E1   -22.067, E3 -437069.476}
SPL {X  -159.990, Y  +525.349, Z    +0.000, E1   -22.050, E3 -437080.317}
SPL {X  -159.990, Y  +523.717, Z    +0.000, E1   -22.050, E3 -437088.883}
SPL {X  -159.990, Y  +521.599, Z    +0.000, E1   -22.060, E3 -437099.951}
SPL {X  -159.990, Y  +519.209, Z    +0.000, E1   -22.063, E3 -437112.425}
SPL {X  -159.990, Y  +517.330, Z    +0.000, E1   -22.053, E3 -437122.281}
SPL {X  -159.990, Y  +514.729, Z    +0.000, E1   -22.089, E3 -437135.839}
SPL {X  -159.990, Y  +511.670, Z    +0.000, E1   -22.064, E3 -437151.927}
SPL {X  -159.990, Y  +506.947, Z    +0.000, E1   -23.726, E3 -437161.955}
SPL {X  -159.990, Y  +496.921, Z    +0.000, E1   -28.340, E3 -437170.704}
SPL {X  -159.990, Y  +495.822, Z    +0.000, E1   -27.449, E3 -437181.452}
SPL {X  -159.990, Y  +494.952, Z    +0.000, E1   -26.628, E3 -437191.035}
SPL {X  -159.990, Y  +493.896, Z    +0.000, E1   -25.736, E3 -437202.365}
SPL {X  -159.990, Y  +491.647, Z    +0.000, E1   -25.401, E3 -437214.900}
SPL {X  -159.990, Y  +488.807, Z    +0.000, E1   -25.397, E3 -437227.599}
SPL {X  -159.990, Y  +486.070, Z    +0.000, E1   -25.399, E3 -437239.830}
SPL {X  -159.990, Y  +482.821, Z    +0.000, E1   -25.411, E3 -437254.331}
SPL {X  -159.990, Y  +480.183, Z    +0.000, E1   -25.384, E3 -437266.171}
SPL {X  -159.990, Y  +477.508, Z    +0.000, E1   -25.410, E3 -437278.080}
SPL {X  -159.990, Y  +473.634, Z    +0.000, E1   -25.426, E3 -437295.369}
SPL {X  -159.990, Y  +470.047, Z    +0.000, E1   -25.402, E3 -437311.450}
SPL {X  -159.990, Y  +466.213, Z    +0.000, E1   -25.433, E3 -437328.530}
SPL {X  -159.990, Y  +462.520, Z    +0.000, E1   -25.400, E3 -437345.098}
SPL {X  -159.990, Y  +460.081, Z    +0.000, E1   -25.390, E3 -437356.000}
SPL {X  -159.990, Y  +457.497, Z    +0.000, E1   -25.403, E3 -437367.524}
SPL {X  -159.990, Y  +454.323, Z    +0.000, E1   -25.412, E3 -437381.684}
SPL {X  -159.990, Y  +451.400, Z    +0.000, E1   -25.397, E3 -437394.774}
SPL {X  -159.990, Y  +448.503, Z    +0.000, E1   -25.410, E3 -437407.692}
SPL {X  -159.990, Y  +445.108, Z    +0.000, E1   -25.407, E3 -437422.930}
SPL {X  -159.990, Y  +441.797, Z    +0.000, E1   -25.390, E3 -437437.809}
SPL {X  -159.990, Y  +439.442, Z    +0.000, E1   -25.369, E3 -437448.386}
SPL {X  -159.990, Y  +436.316, Z    +0.000, E1   -25.420, E3 -437462.268}
SPL {X  -159.990, Y  +432.613, Z    +0.000, E1   -25.390, E3 -437478.893}
SPL {X  -159.990, Y  +429.079, Z    +0.000, E1   -25.407, E3 -437494.664}
SPL {X  -159.990, Y  +426.149, Z    +0.000, E1   -25.374, E3 -437507.826}
SPL {X  -159.990, Y  +423.417, Z    +0.000, E1   -25.400, E3 -437519.991}
SPL {X  -159.990, Y  +420.283, Z    +0.000, E1   -25.386, E3 -437534.036}
SPL {X  -159.990, Y  +417.514, Z    +0.000, E1   -25.386, E3 -437546.420}
SPL {X  -159.990, Y  +414.805, Z    +0.000, E1   -25.385, E3 -437558.540}
SPL {X  -159.990, Y  +411.282, Z    +0.000, E1   -25.413, E3 -437574.241}
SPL {X  -159.990, Y  +407.450, Z    +0.000, E1   -25.401, E3 -437591.390}
SPL {X  -159.990, Y  +403.513, Z    +0.000, E1   -25.420, E3 -437608.944}
SPL {X  -159.990, Y  +399.257, Z    +0.000, E1   -25.420, E3 -437627.985}
SPL {X  -159.990, Y  +395.992, Z    +0.000, E1   -25.380, E3 -437642.674}
SPL {X  -159.990, Y  +393.569, Z    +0.000, E1   -25.379, E3 -437653.518}
SPL {X  -159.990, Y  +390.564, Z    +0.000, E1   -25.393, E3 -437666.962}
SPL {X  -159.990, Y  +387.503, Z    +0.000, E1   -25.378, E3 -437680.676}
SPL {X  -159.990, Y  +384.900, Z    +0.000, E1   -25.383, E3 -437692.286}
SPL {X  -159.990, Y  +382.110, Z    +0.000, E1   -25.393, E3 -437704.733}
SPL {X  -159.961, Y  +379.439, Z    +0.000, E1   -25.380, E3 -437716.712}
SPL {X  -159.894, Y  +376.959, Z    +0.000, E1   -25.370, E3 -437727.889}
SPL {X  -159.784, Y  +374.382, Z    +0.000, E1   -25.356, E3 -437739.530}
SPL {X  -159.621, Y  +371.640, Z    +0.000, E1   -25.335, E3 -437751.970}
SPL {X  -159.406, Y  +368.844, Z    +0.000, E1   -25.307, E3 -437764.683}
SPL {X  -159.144, Y  +366.072, Z    +0.000, E1   -25.281, E3 -437777.290}
SPL {X  -158.822, Y  +363.200, Z    +0.000, E1   -25.236, E3 -437790.463}
SPL {X  -158.491, Y  +360.654, Z    +0.000, E1   -25.188, E3 -437802.203}
SPL {X  -158.127, Y  +358.155, Z    +0.000, E1   -25.126, E3 -437813.823}
SPL {X  -158.095, Y  +357.947, Z    +0.000, E1   -21.741, E3 -437845.395}
ENDSPLINE

SPLINE
SPL {X  -158.454, Y  +360.384, Z    +0.000, E1   -19.366, E3 -437857.546}
SPL {X  -159.737, Y  +373.507, Z    +0.000, E1   -10.311, E3 -437879.582}
SPL {X  -159.990, Y  +382.574, Z    +0.000, E1    -4.463, E3 -437886.269}
SPL {X  -159.990, Y  +387.496, Z    +0.000, E1    -1.004, E3 -437889.014}
SPL {X  -159.990, Y  +395.121, Z    +0.000, E1    +4.514, E3 -437893.327}
SPL {X  -159.990, Y  +407.941, Z    +0.000, E1   +14.126, E3 -437905.401}
SPL {X  -159.990, Y  +418.671, Z    +0.000, E1   +19.855, E3 -437924.817}
SPL {X  -159.990, Y  +428.534, Z    +0.000, E1   +23.299, E3 -437948.337}
SPL {X  -159.990, Y  +430.313, Z    +0.000, E1   +23.313, E3 -437957.050}
SPL {X  -159.990, Y  +432.766, Z    +0.000, E1   +23.321, E3 -437969.095}
SPL {X  -159.990, Y  +434.794, Z    +0.000, E1   +23.304, E3 -437979.126}
SPL {X  -159.990, Y  +437.007, Z    +0.000, E1   +23.323, E3 -437989.978}
SPL {X  -159.990, Y  +439.778, Z    +0.000, E1   +23.323, E3 -438003.611}
SPL {X  -159.990, Y  +442.010, Z    +0.000, E1   +23.308, E3 -438014.632}
SPL {X  -159.990, Y  +443.729, Z    +0.000, E1   +23.310, E3 -438023.088}
SPL {X  -159.990, Y  +446.037, Z    +0.000, E1   +23.324, E3 -438034.425}
SPL {X  -159.990, Y  +449.434, Z    +0.000, E1   +23.356, E3 -438051.046}
SPL {X  -159.990, Y  +453.256, Z    +0.000, E1   +23.349, E3 -438069.881}
SPL {X  -159.990, Y  +455.953, Z    +0.000, E1   +23.320, E3 -438083.196}
SPL {X  -159.990, Y  +458.265, Z    +0.000, E1   +23.328, E3 -438094.550}
SPL {X  -159.990, Y  +461.258, Z    +0.000, E1   +23.344, E3 -438109.266}
SPL {X  -159.990, Y  +464.382, Z    +0.000, E1   +23.332, E3 -438124.647}
SPL {X  -159.990, Y  +466.881, Z    +0.000, E1   +23.322, E3 -438136.967}
SPL {X  -159.990, Y  +468.951, Z    +0.000, E1   +23.319, E3 -438147.159}
SPL {X  -159.990, Y  +470.991, Z    +0.000, E1   +23.322, E3 -438157.189}
SPL {X  -159.990, Y  +474.027, Z    +0.000, E1   +23.352, E3 -438172.093}
SPL {X  -159.990, Y  +477.600, Z    +0.000, E1   +23.351, E3 -438189.697}
SPL {X  -159.990, Y  +481.169, Z    +0.000, E1   +23.337, E3 -438207.294}
SPL {X  -159.990, Y  +483.782, Z    +0.000, E1   +23.316, E3 -438220.199}
SPL {X  -159.990, Y  +486.109, Z    +0.000, E1   +23.322, E3 -438231.651}
SPL {X  -159.990, Y  +489.247, Z    +0.000, E1   +23.348, E3 -438247.038}
SPL {X  -159.990, Y  +492.126, Z    +0.000, E1   +23.317, E3 -438261.273}
SPL {X  -159.990, Y  +494.937, Z    +0.000, E1   +23.343, E3 -438275.055}
SPL {X  -159.990, Y  +497.668, Z    +0.000, E1   +23.317, E3 -438288.548}
SPL {X  -159.990, Y  +499.995, Z    +0.000, E1   +23.324, E3 -438299.986}
SPL {X  -159.990, Y  +502.456, Z    +0.000, E1   +23.324, E3 -438312.100}
SPL {X  -159.990, Y  +504.508, Z    +0.000, E1   +23.311, E3 -438322.235}
SPL {X  -159.990, Y  +506.420, Z    +0.000, E1   +23.317, E3 -438331.627}
SPL {X  -159.990, Y  +508.862, Z    +0.000, E1   +23.328, E3 -438343.620}
SPL {X  -159.990, Y  +511.771, Z    +0.000, E1   +23.331, E3 -438357.942}
SPL {X  -159.990, Y  +514.757, Z    +0.000, E1   +23.329, E3 -438372.650}
SPL {X  -159.990, Y  +517.536, Z    +0.000, E1   +23.326, E3 -438386.316}
SPL {X  -159.990, Y  +519.961, Z    +0.000, E1   +23.334, E3 -438398.169}
SPL {X  -159.990, Y  +521.849, Z    +0.000, E1   +23.320, E3 -438407.491}
SPL {X  -159.990, Y  +523.968, Z    +0.000, E1   +23.332, E3 -438417.927}
SPL {X  -159.990, Y  +526.466, Z    +0.000, E1   +23.320, E3 -438430.270}
SPL {X  -159.990, Y  +528.815, Z    +0.000, E1   +23.322, E3 -438441.830}
SPL {X  -159.990, Y  +531.246, Z    +0.000, E1   +23.325, E3 -438453.768}
SPL {X  -159.990, Y  +533.354, Z    +0.000, E1   +23.318, E3 -438464.154}
SPL {X  -159.990, Y  +534.931, Z    +0.000, E1   +23.312, E3 -438471.948}
SPL {X  -159.990, Y  +537.024, Z    +0.000, E1   +23.321, E3 -438482.247}
SPL {X  -159.990, Y  +539.129, Z    +0.000, E1   +23.310, E3 -438492.630}
SPL {X  -159.990, Y  +541.183, Z    +0.000, E1   +23.319, E3 -438502.727}
SPL {X  -159.990, Y  +544.314, Z    +0.000, E1   +23.352, E3 -438518.055}
SPL {X  -159.990, Y  +548.126, Z    +0.000, E1   +23.354, E3 -438536.810}
SPL {X  -159.990, Y  +551.344, Z    +0.000, E1   +23.327, E3 -438552.702}
SPL {X  -159.990, Y  +553.642, Z    +0.000, E1   +23.319, E3 -438564.021}
SPL {X  -159.990, Y  +556.481, Z    +0.000, E1   +23.354, E3 -438577.928}
SPL {X  -159.990, Y  +559.475, Z    +0.000, E1   +23.321, E3 -438592.733}
SPL {X  -159.990, Y  +561.830, Z    +0.000, E1   +23.325, E3 -438604.318}
SPL {X  -159.990, Y  +564.273, Z    +0.000, E1   +23.325, E3 -438616.342}
SPL {X  -159.990, Y  +566.342, Z    +0.000, E1   +23.314, E3 -438626.547}
SPL {X  -159.990, Y  +568.849, Z    +0.000, E1   +23.338, E3 -438638.842}
SPL {X  -159.990, Y  +572.204, Z    +0.000, E1   +23.344, E3 -438655.337}
SPL {X  -159.990, Y  +575.097, Z    +0.000, E1   +23.325, E3 -438669.613}
SPL {X  -159.990, Y  +577.540, Z    +0.000, E1   +23.325, E3 -438681.642}
SPL {X  -159.990, Y  +580.312, Z    +0.000, E1   +23.340, E3 -438695.224}
SPL {X  -159.990, Y  +583.018, Z    +0.000, E1   +23.331, E3 -438708.529}
SPL {X  -159.990, Y  +585.165, Z    +0.000, E1   +23.322, E3 -438719.145}
SPL {X  -159.990, Y  +587.388, Z    +0.000, E1   +23.328, E3 -438730.057}
SPL {X  -159.990, Y  +589.763, Z    +0.000, E1   +23.328, E3 -438741.744}
SPL {X  -159.990, Y  +592.397, Z    +0.000, E1   +23.344, E3 -438754.625}
SPL {X  -159.990, Y  +594.928, Z    +0.000, E1   +23.334, E3 -438767.087}
SPL {X  -159.990, Y  +597.981, Z    +0.000, E1   +23.373, E3 -438782.002}
SPL {X  -159.990, Y  +600.935, Z    +0.000, E1   +23.343, E3 -438796.534}
SPL {X  -159.990, Y  +603.047, Z    +0.000, E1   +23.344, E3 -438806.920}
SPL {X  -159.990, Y  +605.187, Z    +0.000, E1   +23.344, E3 -438817.442}
SPL {X  -159.990, Y  +607.319, Z    +0.000, E1   +23.353, E3 -438827.904}
SPL {X  -159.990, Y  +610.569, Z    +0.000, E1   +23.372, E3 -438843.869}
SPL {X  -159.990, Y  +613.591, Z    +0.000, E1   +23.342, E3 -438858.798}
SPL {X  -159.990, Y  +615.604, Z    +0.000, E1   +23.330, E3 -438868.736}
SPL {X  -159.990, Y  +618.445, Z    +0.000, E1   +23.368, E3 -438882.649}
SPL {X  -159.990, Y  +621.517, Z    +0.000, E1   +23.337, E3 -438897.813}
SPL {X  -159.990, Y  +623.764, Z    +0.000, E1   +23.335, E3 -438908.863}
SPL {X  -159.990, Y  +625.941, Z    +0.000, E1   +23.337, E3 -438919.555}
SPL {X  -159.990, Y  +628.611, Z    +0.000, E1   +23.357, E3 -438932.634}
SPL {X  -159.990, Y  +631.169, Z    +0.000, E1   +23.338, E3 -438945.238}
SPL {X  -159.990, Y  +633.318, Z    +0.000, E1   +23.339, E3 -438955.827}
SPL {X  -159.990, Y  +635.650, Z    +0.000, E1   +23.339, E3 -438967.298}
SPL {X  -159.990, Y  +637.839, Z    +0.000, E1   +23.335, E3 -438978.108}
SPL {X  -159.990, Y  +640.072, Z    +0.000, E1   +23.325, E3 -438989.140}
SPL {X  -159.990, Y  +642.230, Z    +0.000, E1   +23.323, E3 -438999.822}
SPL {X  -159.990, Y  +645.287, Z    +0.000, E1   +23.340, E3 -439014.848}
SPL {X  -159.990, Y  +648.792, Z    +0.000, E1   +23.346, E3 -439032.107}
SPL {X  -159.990, Y  +651.647, Z    +0.000, E1   +23.312, E3 -439046.219}
SPL {X  -159.990, Y  +654.543, Z    +0.000, E1   +23.348, E3 -439060.385}
SPL {X  -159.990, Y  +658.319, Z    +0.000, E1   +23.349, E3 -439078.975}
SPL {X  -159.990, Y  +661.392, Z    +0.000, E1   +23.318, E3 -439094.178}
SPL {X  -159.990, Y  +663.662, Z    +0.000, E1   +23.322, E3 -439105.302}
SPL {X  -159.990, Y  +665.964, Z    +0.000, E1   +23.328, E3 -439116.592}
SPL {X  -159.990, Y  +667.870, Z    +0.000, E1   +23.320, E3 -439125.999}
SPL {X  -159.990, Y  +669.861, Z    +0.000, E1   +23.321, E3 -439135.800}
SPL {X  -159.983, Y  +672.946, Z    +0.000, E1   +23.359, E3 -439150.910}
SPL {X  -159.924, Y  +676.110, Z    +0.000, E1   +23.320, E3 -439166.609}
SPL {X  -159.845, Y  +678.302, Z    +0.000, E1   +23.298, E3 -439177.511}
SPL {X  -159.760, Y  +680.081, Z    +0.000, E1   +23.288, E3 -439186.354}
SPL {X  -159.626, Y  +682.287, Z    +0.000, E1   +23.280, E3 -439197.326}
SPL {X  -159.462, Y  +684.486, Z    +0.000, E1   +23.258, E3 -439208.325}
SPL {X  -159.246, Y  +686.911, Z    +0.000, E1   +23.230, E3 -439220.487}
SPL {X  -159.019, Y  +689.098, Z    +0.000, E1   +23.200, E3 -439231.489}
SPL {X  -158.771, Y  +691.210, Z    +0.000, E1   +23.159, E3 -439242.164}
SPL {X  -158.553, Y  +692.896, Z    +0.000, E1   +23.130, E3 -439250.693}
ENDSPLINE

SPLINE
SPL {X  -159.063, Y  +688.696, Z    +0.000, E1   +17.094, E3 -439288.814}
SPL {X  -159.987, Y  +672.488, Z    +0.000, E1    +5.638, E3 -439312.879}
SPL {X  -159.990, Y  +663.928, Z    +0.000, E1    -0.338, E3 -439318.674}
SPL {X  -159.990, Y  +658.009, Z    +0.000, E1    -4.774, E3 -439322.374}
SPL {X  -159.990, Y  +651.567, Z    +0.000, E1    -9.674, E3 -439327.777}
SPL {X  -159.990, Y  +637.762, Z    +0.000, E1   -18.345, E3 -439345.135}
SPL {X  -159.990, Y  +626.382, Z    +0.000, E1   -22.040, E3 -439377.184}
SPL {X  -159.990, Y  +623.760, Z    +0.000, E1   -22.031, E3 -439390.962}
SPL {X  -159.990, Y  +621.334, Z    +0.000, E1   -22.029, E3 -439403.688}
SPL {X  -159.990, Y  +618.387, Z    +0.000, E1   -22.057, E3 -439419.078}
SPL {X  -159.990, Y  +615.830, Z    +0.000, E1   -22.023, E3 -439432.569}
SPL {X  -159.990, Y  +613.034, Z    +0.000, E1   -22.053, E3 -439447.176}
SPL {X  -159.990, Y  +609.503, Z    +0.000, E1   -22.054, E3 -439465.703}
SPL {X  -159.990, Y  +605.804, Z    +0.000, E1   -22.064, E3 -439485.047}
SPL {X  -159.990, Y  +602.819, Z    +0.000, E1   -22.037, E3 -439500.718}
SPL {X  -159.990, Y  +600.642, Z    +0.000, E1   -22.032, E3 -439512.146}
SPL {X  -159.990, Y  +598.568, Z    +0.000, E1   -22.046, E3 -439522.939}
SPL {X  -159.990, Y  +595.493, Z    +0.000, E1   -22.070, E3 -439539.022}
SPL {X  -159.990, Y  +592.865, Z    +0.000, E1   -22.036, E3 -439552.851}
SPL {X  -159.990, Y  +590.803, Z    +0.000, E1   -22.046, E3 -439563.641}
SPL {X  -159.990, Y  +587.778, Z    +0.000, E1   -22.073, E3 -439579.417}
SPL {X  -159.990, Y  +585.120, Z    +0.000, E1   -22.045, E3 -439593.361}
SPL {X  -159.990, Y  +583.118, Z    +0.000, E1   -22.052, E3 -439603.847}
SPL {X  -159.990, Y  +580.131, Z    +0.000, E1   -22.078, E3 -439619.453}
SPL {X  -159.990, Y  +576.888, Z    +0.000, E1   -22.061, E3 -439636.483}
SPL {X  -159.990, Y  +574.280, Z    +0.000, E1   -22.051, E3 -439650.157}
SPL {X  -159.990, Y  +572.375, Z    +0.000, E1   -22.037, E3 -439660.196}
SPL {X  -159.990, Y  +569.881, Z    +0.000, E1   -22.067, E3 -439673.190}
SPL {X  -159.990, Y  +567.211, Z    +0.000, E1   -22.046, E3 -439687.217}
SPL {X  -159.990, Y  +565.039, Z    +0.000, E1   -22.047, E3 -439698.595}
SPL {X  -159.990, Y  +562.755, Z    +0.000, E1   -22.047, E3 -439710.580}
SPL {X  -159.990, Y  +559.661, Z    +0.000, E1   -22.078, E3 -439726.712}
SPL {X  -159.990, Y  +555.965, Z    +0.000, E1   -22.085, E3 -439746.021}
SPL {X  -159.990, Y  +553.115, Z    +0.000, E1   -22.054, E3 -439761.006}
SPL {X  -159.990, Y  +550.886, Z    +0.000, E1   -22.056, E3 -439772.688}
SPL {X  -159.990, Y  +547.986, Z    +0.000, E1   -22.078, E3 -439787.807}
SPL {X  -159.990, Y  +545.350, Z    +0.000, E1   -22.053, E3 -439801.668}
SPL {X  -159.990, Y  +543.405, Z    +0.000, E1   -22.048, E3 -439811.881}
SPL {X  -159.990, Y  +541.673, Z    +0.000, E1   -22.053, E3 -439820.945}
SPL {X  -159.990, Y  +539.341, Z    +0.000, E1   -22.056, E3 -439833.150}
SPL {X  -159.990, Y  +536.301, Z    +0.000, E1   -22.084, E3 -439849.005}
SPL {X  -159.990, Y  +533.389, Z    +0.000, E1   -22.057, E3 -439864.312}
SPL {X  -159.990, Y  +531.347, Z    +0.000, E1   -22.052, E3 -439875.013}
SPL {X  -159.990, Y  +528.972, Z    +0.000, E1   -22.072, E3 -439887.386}
SPL {X  -159.990, Y  +526.034, Z    +0.000, E1   -22.073, E3 -439902.765}
SPL {X  -159.990, Y  +523.717, Z    +0.000, E1   -22.050, E3 -439914.970}
SPL {X  -159.990, Y  +521.599, Z    +0.000, E1   -22.060, E3 -439926.038}
SPL {X  -159.990, Y  +519.209, Z    +0.000, E1   -22.063, E3 -439938.512}
SPL {X  -159.990, Y  +517.330, Z    +0.000, E1   -22.053, E3 -439948.368}
SPL {X  -159.990, Y  +514.729, Z    +0.000, E1   -22.089, E3 -439961.926}
SPL {X  -159.990, Y  +511.670, Z    +0.000, E1   -22.064, E3 -439978.014}
SPL {X  -159.990, Y  +506.947, Z    +0.000, E1   -23.726, E3 -439988.042}
SPL {X  -159.990, Y  +496.921, Z    +0.000, E1   -28.340, E3 -439996.791}
SPL {X  -159.990, Y  +495.822, Z    +0.000, E1   -27.449, E3 -440007.539}
SPL {X  -159.990, Y  +494.952, Z    +0.000, E1   -26.628, E3 -440017.122}
SPL {X  -159.990, Y  +493.896, Z    +0.000, E1   -25.736, E3 -440028.452}
SPL {X  -159.990, Y  +491.647, Z    +0.000, E1   -25.401, E3 -440040.987}
SPL {X  -159.990, Y  +488.807, Z    +0.000, E1   -25.397, E3 -440053.686}
SPL {X  -159.990, Y  +486.070, Z    +0.000, E1   -25.399, E3 -440065.917}
SPL {X  -159.990, Y  +483.747, Z    +0.000, E1   -25.384, E3 -440076.329}
SPL {X  -159.990, Y  +481.038, Z    +0.000, E1   -25.412, E3 -440088.385}
SPL {X  -159.990, Y  +477.508, Z    +0.000, E1   -25.410, E3 -440104.167}
SPL {X  -159.990, Y  +473.634, Z    +0.000, E1   -25.426, E3 -440121.456}
SPL {X  -159.990, Y  +470.047, Z    +0.000, E1   -25.402, E3 -440137.537}
SPL {X  -159.990, Y  +467.082, Z    +0.000, E1   -25.399, E3 -440150.784}
SPL {X  -159.990, Y  +464.063, Z    +0.000, E1   -25.405, E3 -440164.279}
SPL {X  -159.990, Y  +460.712, Z    +0.000, E1   -25.411, E3 -440179.239}
SPL {X  -159.990, Y  +457.497, Z    +0.000, E1   -25.403, E3 -440193.611}
SPL {X  -159.990, Y  +454.323, Z    +0.000, E1   -25.412, E3 -440207.771}
SPL {X  -159.990, Y  +450.823, Z    +0.000, E1   -25.417, E3 -440223.399}
SPL {X  -159.990, Y  +447.982, Z    +0.000, E1   -25.393, E3 -440236.140}
SPL {X  -159.990, Y  +445.108, Z    +0.000, E1   -25.407, E3 -440249.017}
SPL {X  -159.990, Y  +441.797, Z    +0.000, E1   -25.390, E3 -440263.896}
SPL {X  -159.990, Y  +439.442, Z    +0.000, E1   -25.369, E3 -440274.473}
SPL {X  -159.990, Y  +436.316, Z    +0.000, E1   -25.420, E3 -440288.355}
SPL {X  -159.990, Y  +432.613, Z    +0.000, E1   -25.390, E3 -440304.980}
SPL {X  -159.990, Y  +429.827, Z    +0.000, E1   -25.380, E3 -440317.457}
SPL {X  -159.990, Y  +426.865, Z    +0.000, E1   -25.398, E3 -440330.662}
SPL {X  -159.990, Y  +423.417, Z    +0.000, E1   -25.400, E3 -440346.078}
SPL {X  -159.990, Y  +420.283, Z    +0.000, E1   -25.386, E3 -440360.123}
SPL {X  -159.990, Y  +417.514, Z    +0.000, E1   -25.386, E3 -440372.507}
SPL {X  -159.990, Y  +414.805, Z    +0.000, E1   -25.385, E3 -440384.627}
SPL {X  -159.990, Y  +411.959, Z    +0.000, E1   -25.386, E3 -440397.354}
SPL {X  -159.990, Y  +408.981, Z    +0.000, E1   -25.392, E3 -440410.658}
SPL {X  -159.990, Y  +405.773, Z    +0.000, E1   -25.398, E3 -440424.968}
SPL {X  -159.990, Y  +402.805, Z    +0.000, E1   -25.389, E3 -440438.254}
SPL {X  -159.990, Y  +400.083, Z    +0.000, E1   -25.388, E3 -440450.430}
SPL {X  -159.990, Y  +396.740, Z    +0.000, E1   -25.410, E3 -440465.355}
SPL {X  -159.990, Y  +393.569, Z    +0.000, E1   -25.379, E3 -440479.605}
SPL {X  -159.990, Y  +390.564, Z    +0.000, E1   -25.393, E3 -440493.049}
SPL {X  -159.990, Y  +387.503, Z    +0.000, E1   -25.378, E3 -440506.763}
SPL {X  -159.990, Y  +384.900, Z    +0.000, E1   -25.383, E3 -440518.373}
SPL {X  -159.990, Y  +382.110, Z    +0.000, E1   -25.393, E3 -440530.820}
SPL {X  -159.961, Y  +379.439, Z    +0.000, E1   -25.380, E3 -440542.799}
SPL {X  -159.894, Y  +376.959, Z    +0.000, E1   -25.370, E3 -440553.976}
SPL {X  -159.784, Y  +374.382, Z    +0.000, E1   -25.356, E3 -440565.617}
SPL {X  -159.621, Y  +371.640, Z    +0.000, E1   -25.335, E3 -440578.057}
SPL {X  -159.406, Y  +368.844, Z    +0.000, E1   -25.307, E3 -440590.770}
SPL {X  -159.144, Y  +366.072, Z    +0.000, E1   -25.281, E3 -440603.377}
SPL {X  -158.822, Y  +363.200, Z    +0.000, E1   -25.236, E3 -440616.550}
SPL {X  -158.491, Y  +360.654, Z    +0.000, E1   -25.188, E3 -440628.290}
SPL {X  -158.127, Y  +358.155, Z    +0.000, E1   -25.126, E3 -440639.910}
SPL {X  -158.095, Y  +357.947, Z    +0.000, E1   -21.741, E3 -440671.482}
ENDSPLINE

SPLINE
SPL {X  -158.454, Y  +360.384, Z    +0.000, E1   -19.366, E3 -440683.633}
SPL {X  -159.737, Y  +373.507, Z    +0.000, E1   -10.311, E3 -440705.668}
SPL {X  -159.990, Y  +382.574, Z    +0.000, E1    -4.463, E3 -440712.356}
SPL {X  -159.990, Y  +387.496, Z    +0.000, E1    -1.004, E3 -440715.101}
SPL {X  -159.990, Y  +395.121, Z    +0.000, E1    +4.514, E3 -440719.414}
SPL {X  -159.990, Y  +407.941, Z    +0.000, E1   +14.126, E3 -440731.488}
SPL {X  -159.990, Y  +418.671, Z    +0.000, E1   +19.855, E3 -440750.904}
SPL {X  -159.990, Y  +429.878, Z    +0.000, E1   +23.330, E3 -440780.959}
SPL {X  -159.990, Y  +432.766, Z    +0.000, E1   +23.321, E3 -440795.182}
SPL {X  -159.990, Y  +434.794, Z    +0.000, E1   +23.304, E3 -440805.213}
SPL {X  -159.990, Y  +437.007, Z    +0.000, E1   +23.323, E3 -440816.065}
SPL {X  -159.990, Y  +439.778, Z    +0.000, E1   +23.323, E3 -440829.698}
SPL {X  -159.990, Y  +442.945, Z    +0.000, E1   +23.339, E3 -440845.262}
SPL {X  -159.990, Y  +446.037, Z    +0.000, E1   +23.324, E3 -440860.512}
SPL {X  -159.990, Y  +448.797, Z    +0.000, E1   +23.331, E3 -440874.042}
SPL {X  -159.990, Y  +451.747, Z    +0.000, E1   +23.333, E3 -440888.590}
SPL {X  -159.990, Y  +454.210, Z    +0.000, E1   +23.316, E3 -440900.721}
SPL {X  -159.990, Y  +455.953, Z    +0.000, E1   +23.320, E3 -440909.282}
SPL {X  -159.990, Y  +458.265, Z    +0.000, E1   +23.328, E3 -440920.637}
SPL {X  -159.990, Y  +460.492, Z    +0.000, E1   +23.317, E3 -440931.636}
SPL {X  -159.990, Y  +462.929, Z    +0.000, E1   +23.331, E3 -440943.592}
SPL {X  -159.990, Y  +466.197, Z    +0.000, E1   +23.351, E3 -440959.629}
SPL {X  -159.990, Y  +468.951, Z    +0.000, E1   +23.319, E3 -440973.246}
SPL {X  -159.990, Y  +470.991, Z    +0.000, E1   +23.322, E3 -440983.276}
SPL {X  -159.990, Y  +474.027, Z    +0.000, E1   +23.352, E3 -440998.180}
SPL {X  -159.990, Y  +476.830, Z    +0.000, E1   +23.323, E3 -441012.048}
SPL {X  -159.990, Y  +479.553, Z    +0.000, E1   +23.328, E3 -441025.450}
SPL {X  -159.990, Y  +482.950, Z    +0.000, E1   +23.350, E3 -441042.122}
SPL {X  -159.990, Y  +486.109, Z    +0.000, E1   +23.322, E3 -441057.738}
SPL {X  -159.990, Y  +488.481, Z    +0.000, E1   +23.319, E3 -441069.418}
SPL {X  -159.990, Y  +491.454, Z    +0.000, E1   +23.343, E3 -441083.998}
SPL {X  -159.990, Y  +494.937, Z    +0.000, E1   +23.343, E3 -441101.142}
SPL {X  -159.990, Y  +497.668, Z    +0.000, E1   +23.317, E3 -441114.635}
SPL {X  -159.990, Y  +499.995, Z    +0.000, E1   +23.324, E3 -441126.073}
SPL {X  -159.990, Y  +502.456, Z    +0.000, E1   +23.324, E3 -441138.187}
SPL {X  -159.990, Y  +504.508, Z    +0.000, E1   +23.311, E3 -441148.321}
SPL {X  -159.990, Y  +506.420, Z    +0.000, E1   +23.317, E3 -441157.714}
SPL {X  -159.990, Y  +508.862, Z    +0.000, E1   +23.328, E3 -441169.707}
SPL {X  -159.990, Y  +511.771, Z    +0.000, E1   +23.331, E3 -441184.029}
SPL {X  -159.990, Y  +514.016, Z    +0.000, E1   +23.308, E3 -441195.133}
SPL {X  -159.990, Y  +516.860, Z    +0.000, E1   +23.355, E3 -441209.019}
SPL {X  -159.990, Y  +520.719, Z    +0.000, E1   +23.363, E3 -441227.929}
SPL {X  -159.990, Y  +523.968, Z    +0.000, E1   +23.332, E3 -441244.014}
SPL {X  -159.990, Y  +526.466, Z    +0.000, E1   +23.320, E3 -441256.357}
SPL {X  -159.990, Y  +528.815, Z    +0.000, E1   +23.322, E3 -441267.917}
SPL {X  -159.990, Y  +531.246, Z    +0.000, E1   +23.325, E3 -441279.855}
SPL {X  -159.990, Y  +533.354, Z    +0.000, E1   +23.318, E3 -441290.241}
SPL {X  -159.990, Y  +534.931, Z    +0.000, E1   +23.312, E3 -441298.035}
SPL {X  -159.990, Y  +537.024, Z    +0.000, E1   +23.321, E3 -441308.334}
SPL {X  -159.990, Y  +539.129, Z    +0.000, E1   +23.310, E3 -441318.717}
SPL {X  -159.990, Y  +541.183, Z    +0.000, E1   +23.319, E3 -441328.814}
SPL {X  -159.990, Y  +544.314, Z    +0.000, E1   +23.352, E3 -441344.142}
SPL {X  -159.990, Y  +548.126, Z    +0.000, E1   +23.354, E3 -441362.897}
SPL {X  -159.990, Y  +551.344, Z    +0.000, E1   +23.327, E3 -441378.789}
SPL {X  -159.990, Y  +553.642, Z    +0.000, E1   +23.319, E3 -441390.108}
SPL {X  -159.990, Y  +556.481, Z    +0.000, E1   +23.354, E3 -441404.015}
SPL {X  -159.990, Y  +559.475, Z    +0.000, E1   +23.321, E3 -441418.820}
SPL {X  -159.990, Y  +561.830, Z    +0.000, E1   +23.325, E3 -441430.405}
SPL {X  -159.990, Y  +564.273, Z    +0.000, E1   +23.325, E3 -441442.429}
SPL {X  -159.990, Y  +567.351, Z    +0.000, E1   +23.348, E3 -441457.525}
SPL {X  -159.990, Y  +570.560, Z    +0.000, E1   +23.333, E3 -441473.354}
SPL {X  -159.990, Y  +572.975, Z    +0.000, E1   +23.316, E3 -441485.274}
SPL {X  -159.990, Y  +575.097, Z    +0.000, E1   +23.325, E3 -441495.700}
SPL {X  -159.990, Y  +577.540, Z    +0.000, E1   +23.325, E3 -441507.729}
SPL {X  -159.990, Y  +580.312, Z    +0.000, E1   +23.340, E3 -441521.311}
SPL {X  -159.990, Y  +583.018, Z    +0.000, E1   +23.331, E3 -441534.616}
SPL {X  -159.990, Y  +585.165, Z    +0.000, E1   +23.322, E3 -441545.231}
SPL {X  -159.990, Y  +587.388, Z    +0.000, E1   +23.328, E3 -441556.144}
SPL {X  -159.990, Y  +589.763, Z    +0.000, E1   +23.328, E3 -441567.831}
SPL {X  -159.990, Y  +592.397, Z    +0.000, E1   +23.344, E3 -441580.712}
SPL {X  -159.990, Y  +595.589, Z    +0.000, E1   +23.356, E3 -441596.385}
SPL {X  -159.990, Y  +598.571, Z    +0.000, E1   +23.347, E3 -441611.028}
SPL {X  -159.990, Y  +600.935, Z    +0.000, E1   +23.343, E3 -441622.621}
SPL {X  -159.990, Y  +603.047, Z    +0.000, E1   +23.344, E3 -441633.007}
SPL {X  -159.990, Y  +605.187, Z    +0.000, E1   +23.344, E3 -441643.529}
SPL {X  -159.990, Y  +607.319, Z    +0.000, E1   +23.353, E3 -441653.991}
SPL {X  -159.990, Y  +609.514, Z    +0.000, E1   +23.337, E3 -441664.820}
SPL {X  -159.990, Y  +611.376, Z    +0.000, E1   +23.336, E3 -441674.008}
SPL {X  -159.990, Y  +613.591, Z    +0.000, E1   +23.342, E3 -441684.885}
SPL {X  -159.990, Y  +615.604, Z    +0.000, E1   +23.330, E3 -441694.823}
SPL {X  -159.990, Y  +617.623, Z    +0.000, E1   +23.337, E3 -441704.753}
SPL {X  -159.990, Y  +620.788, Z    +0.000, E1   +23.368, E3 -441720.258}
SPL {X  -159.990, Y  +623.764, Z    +0.000, E1   +23.335, E3 -441734.950}
SPL {X  -159.990, Y  +625.941, Z    +0.000, E1   +23.337, E3 -441745.642}
SPL {X  -159.990, Y  +628.611, Z    +0.000, E1   +23.357, E3 -441758.720}
SPL {X  -159.990, Y  +631.169, Z    +0.000, E1   +23.338, E3 -441771.325}
SPL {X  -159.990, Y  +633.318, Z    +0.000, E1   +23.339, E3 -441781.914}
SPL {X  -159.990, Y  +635.650, Z    +0.000, E1   +23.339, E3 -441793.385}
SPL {X  -159.990, Y  +637.839, Z    +0.000, E1   +23.335, E3 -441804.195}
SPL {X  -159.990, Y  +640.072, Z    +0.000, E1   +23.325, E3 -441815.227}
SPL {X  -159.990, Y  +642.230, Z    +0.000, E1   +23.323, E3 -441825.909}
SPL {X  -159.990, Y  +645.287, Z    +0.000, E1   +23.340, E3 -441840.935}
SPL {X  -159.990, Y  +648.792, Z    +0.000, E1   +23.346, E3 -441858.193}
SPL {X  -159.990, Y  +652.623, Z    +0.000, E1   +23.348, E3 -441877.028}
SPL {X  -159.990, Y  +656.380, Z    +0.000, E1   +23.347, E3 -441895.523}
SPL {X  -159.990, Y  +659.180, Z    +0.000, E1   +23.314, E3 -441909.371}
SPL {X  -159.990, Y  +661.392, Z    +0.000, E1   +23.318, E3 -441920.265}
SPL {X  -159.990, Y  +663.662, Z    +0.000, E1   +23.322, E3 -441931.389}
SPL {X  -159.990, Y  +665.964, Z    +0.000, E1   +23.328, E3 -441942.679}
SPL {X  -159.990, Y  +668.989, Z    +0.000, E1   +23.359, E3 -441957.515}
SPL {X  -159.983, Y  +672.946, Z    +0.000, E1   +23.359, E3 -441976.997}
SPL {X  -159.924, Y  +676.110, Z    +0.000, E1   +23.320, E3 -441992.696}
SPL {X  -159.845, Y  +678.302, Z    +0.000, E1   +23.298, E3 -442003.598}
SPL {X  -159.760, Y  +680.081, Z    +0.000, E1   +23.288, E3 -442012.441}
SPL {X  -159.626, Y  +682.287, Z    +0.000, E1   +23.280, E3 -442023.413}
SPL {X  -159.462, Y  +684.486, Z    +0.000, E1   +23.258, E3 -442034.412}
SPL {X  -159.246, Y  +686.911, Z    +0.000, E1   +23.230, E3 -442046.574}
SPL {X  -159.019, Y  +689.098, Z    +0.000, E1   +23.200, E3 -442057.576}
SPL {X  -158.660, Y  +692.086, Z    +0.000, E1   +23.176, E3 -442072.620}
ENDSPLINE

SPLINE
SPL {X  -159.063, Y  +688.696, Z    +0.000, E1   +17.094, E3 -442114.901}
SPL {X  -159.987, Y  +672.488, Z    +0.000, E1    +5.638, E3 -442138.966}
SPL {X  -159.990, Y  +663.928, Z    +0.000, E1    -0.338, E3 -442144.761}
SPL {X  -159.990, Y  +658.009, Z    +0.000, E1    -4.774, E3 -442148.461}
SPL {X  -159.990, Y  +651.567, Z    +0.000, E1    -9.674, E3 -442153.864}
SPL {X  -159.990, Y  +637.762, Z    +0.000, E1   -18.345, E3 -442171.222}
SPL {X  -159.990, Y  +626.382, Z    +0.000, E1   -22.040, E3 -442203.271}
SPL {X  -159.990, Y  +623.760, Z    +0.000, E1   -22.031, E3 -442217.049}
SPL {X  -159.990, Y  +621.334, Z    +0.000, E1   -22.029, E3 -442229.775}
SPL {X  -159.990, Y  +618.387, Z    +0.000, E1   -22.057, E3 -442245.165}
SPL {X  -159.990, Y  +614.928, Z    +0.000, E1   -22.055, E3 -442263.318}
SPL {X  -159.990, Y  +611.459, Z    +0.000, E1   -22.053, E3 -442281.521}
SPL {X  -159.990, Y  +608.810, Z    +0.000, E1   -22.023, E3 -442295.489}
SPL {X  -159.990, Y  +606.481, Z    +0.000, E1   -22.033, E3 -442307.664}
SPL {X  -159.990, Y  +603.419, Z    +0.000, E1   -22.064, E3 -442323.604}
SPL {X  -159.990, Y  +600.642, Z    +0.000, E1   -22.032, E3 -442338.233}
SPL {X  -159.990, Y  +598.568, Z    +0.000, E1   -22.046, E3 -442349.026}
SPL {X  -159.990, Y  +595.493, Z    +0.000, E1   -22.070, E3 -442365.109}
SPL {X  -159.990, Y  +592.865, Z    +0.000, E1   -22.036, E3 -442378.938}
SPL {X  -159.990, Y  +590.803, Z    +0.000, E1   -22.046, E3 -442389.728}
SPL {X  -159.990, Y  +587.778, Z    +0.000, E1   -22.073, E3 -442405.504}
SPL {X  -159.990, Y  +585.120, Z    +0.000, E1   -22.045, E3 -442419.448}
SPL {X  -159.990, Y  +583.118, Z    +0.000, E1   -22.052, E3 -442429.934}
SPL {X  -159.990, Y  +580.131, Z    +0.000, E1   -22.078, E3 -442445.540}
SPL {X  -159.990, Y  +576.888, Z    +0.000, E1   -22.061, E3 -442462.570}
SPL {X  -159.990, Y  +574.280, Z    +0.000, E1   -22.051, E3 -442476.244}
SPL {X  -159.990, Y  +572.375, Z    +0.000, E1   -22.037, E3 -442486.283}
SPL {X  -159.990, Y  +569.881, Z    +0.000, E1   -22.067, E3 -442499.277}
SPL {X  -159.990, Y  +567.211, Z    +0.000, E1   -22.046, E3 -442513.304}
SPL {X  -159.990, Y  +565.039, Z    +0.000, E1   -22.047, E3 -442524.682}
SPL {X  -159.990, Y  +562.755, Z    +0.000, E1   -22.047, E3 -442536.667}
SPL {X  -159.990, Y  +559.661, Z    +0.000, E1   -22.078, E3 -442552.799}
SPL {X  -159.990, Y  +555.965, Z    +0.000, E1   -22.085, E3 -442572.107}
SPL {X  -159.990, Y  +553.115, Z    +0.000, E1   -22.054, E3 -442587.093}
SPL {X  -159.990, Y  +550.886, Z    +0.000, E1   -22.056, E3 -442598.775}
SPL {X  -159.990, Y  +547.986, Z    +0.000, E1   -22.078, E3 -442613.894}
SPL {X  -159.990, Y  +545.350, Z    +0.000, E1   -22.053, E3 -442627.755}
SPL {X  -159.990, Y  +543.405, Z    +0.000, E1   -22.048, E3 -442637.968}
SPL {X  -159.990, Y  +541.673, Z    +0.000, E1   -22.053, E3 -442647.032}
SPL {X  -159.990, Y  +539.341, Z    +0.000, E1   -22.056, E3 -442659.237}
SPL {X  -159.990, Y  +536.301, Z    +0.000, E1   -22.084, E3 -442675.092}
SPL {X  -159.990, Y  +533.389, Z    +0.000, E1   -22.057, E3 -442690.399}
SPL {X  -159.990, Y  +531.347, Z    +0.000, E1   -22.052, E3 -442701.100}
SPL {X  -159.990, Y  +529.626, Z    +0.000, E1   -22.051, E3 -442710.097}
SPL {X  -159.990, Y  +527.412, Z    +0.000, E1   -22.067, E3 -442721.650}
SPL {X  -159.990, Y  +524.425, Z    +0.000, E1   -22.078, E3 -442737.282}
SPL {X  -159.990, Y  +521.599, Z    +0.000, E1   -22.060, E3 -442752.125}
SPL {X  -159.990, Y  +519.209, Z    +0.000, E1   -22.063, E3 -442764.599}
SPL {X  -159.990, Y  +516.651, Z    +0.000, E1   -22.071, E3 -442777.979}
SPL {X  -159.990, Y  +514.122, Z    +0.000, E1   -22.061, E3 -442791.251}
SPL {X  -159.990, Y  +511.670, Z    +0.000, E1   -22.064, E3 -442804.101}
SPL {X  -159.990, Y  +506.947, Z    +0.000, E1   -23.726, E3 -442814.129}
SPL {X  -159.990, Y  +496.921, Z    +0.000, E1   -28.340, E3 -442822.878}
SPL {X  -159.990, Y  +495.822, Z    +0.000, E1   -27.449, E3 -442833.626}
SPL {X  -159.990, Y  +494.952, Z    +0.000, E1   -26.628, E3 -442843.209}
SPL {X  -159.990, Y  +493.896, Z    +0.000, E1   -25.736, E3 -442854.539}
SPL {X  -159.990, Y  +491.647, Z    +0.000, E1   -25.401, E3 -442867.074}
SPL {X  -159.990, Y  +488.807, Z    +0.000, E1   -25.397, E3 -442879.773}
SPL {X  -159.990, Y  +486.070, Z    +0.000, E1   -25.399, E3 -442892.004}
SPL {X  -159.990, Y  +483.747, Z    +0.000, E1   -25.384, E3 -442902.416}
SPL {X  -159.990, Y  +481.038, Z    +0.000, E1   -25.412, E3 -442914.472}
SPL {X  -159.990, Y  +478.407, Z    +0.000, E1   -25.384, E3 -442926.286}
SPL {X  -159.990, Y  +475.940, Z    +0.000, E1   -25.403, E3 -442937.276}
SPL {X  -159.990, Y  +473.026, Z    +0.000, E1   -25.399, E3 -442950.306}
SPL {X  -159.990, Y  +470.047, Z    +0.000, E1   -25.402, E3 -442963.624}
SPL {X  -159.990, Y  +466.213, Z    +0.000, E1   -25.433, E3 -442980.704}
SPL {X  -159.990, Y  +462.520, Z    +0.000, E1   -25.400, E3 -442997.272}
SPL {X  -159.990, Y  +460.081, Z    +0.000, E1   -25.390, E3 -443008.174}
SPL {X  -159.990, Y  +457.497, Z    +0.000, E1   -25.403, E3 -443019.698}
SPL {X  -159.990, Y  +455.126, Z    +0.000, E1   -25.389, E3 -443030.307}
SPL {X  -159.990, Y  +453.438, Z    +0.000, E1   -25.385, E3 -443037.867}
SPL {X  -159.990, Y  +450.823, Z    +0.000, E1   -25.417, E3 -443049.486}
SPL {X  -159.990, Y  +446.894, Z    +0.000, E1   -25.428, E3 -443067.043}
SPL {X  -159.990, Y  +443.345, Z    +0.000, E1   -25.390, E3 -443083.051}
SPL {X  -159.990, Y  +441.077, Z    +0.000, E1   -25.369, E3 -443093.249}
SPL {X  -159.990, Y  +438.608, Z    +0.000, E1   -25.392, E3 -443104.246}
SPL {X  -159.990, Y  +434.852, Z    +0.000, E1   -25.415, E3 -443121.000}
SPL {X  -159.990, Y  +431.966, Z    +0.000, E1   -25.371, E3 -443133.998}
SPL {X  -159.990, Y  +429.079, Z    +0.000, E1   -25.407, E3 -443146.838}
SPL {X  -159.990, Y  +426.149, Z    +0.000, E1   -25.374, E3 -443160.000}
SPL {X  -159.990, Y  +423.417, Z    +0.000, E1   -25.400, E3 -443172.165}
SPL {X  -159.990, Y  +420.283, Z    +0.000, E1   -25.386, E3 -443186.210}
SPL {X  -159.990, Y  +417.514, Z    +0.000, E1   -25.386, E3 -443198.594}
SPL {X  -159.990, Y  +414.805, Z    +0.000, E1   -25.385, E3 -443210.714}
SPL {X  -159.990, Y  +411.959, Z    +0.000, E1   -25.386, E3 -443223.441}
SPL {X  -159.990, Y  +408.981, Z    +0.000, E1   -25.392, E3 -443236.745}
SPL {X  -159.990, Y  +405.773, Z    +0.000, E1   -25.398, E3 -443251.055}
SPL {X  -159.990, Y  +402.805, Z    +0.000, E1   -25.389, E3 -443264.341}
SPL {X  -159.990, Y  +400.083, Z    +0.000, E1   -25.388, E3 -443276.517}
SPL {X  -159.990, Y  +396.740, Z    +0.000, E1   -25.410, E3 -443291.442}
SPL {X  -159.990, Y  +393.569, Z    +0.000, E1   -25.379, E3 -443305.692}
SPL {X  -159.990, Y  +390.564, Z    +0.000, E1   -25.393, E3 -443319.136}
SPL {X  -159.990, Y  +387.503, Z    +0.000, E1   -25.378, E3 -443332.850}
SPL {X  -159.990, Y  +384.900, Z    +0.000, E1   -25.383, E3 -443344.460}
SPL {X  -159.990, Y  +382.110, Z    +0.000, E1   -25.393, E3 -443356.906}
SPL {X  -159.961, Y  +379.439, Z    +0.000, E1   -25.380, E3 -443368.886}
SPL {X  -159.894, Y  +376.959, Z    +0.000, E1   -25.370, E3 -443380.063}
SPL {X  -159.784, Y  +374.382, Z    +0.000, E1   -25.356, E3 -443391.704}
SPL {X  -159.621, Y  +371.640, Z    +0.000, E1   -25.335, E3 -443404.144}
SPL {X  -159.406, Y  +368.844, Z    +0.000, E1   -25.307, E3 -443416.857}
SPL {X  -159.144, Y  +366.072, Z    +0.000, E1   -25.281, E3 -443429.464}
SPL {X  -158.822, Y  +363.200, Z    +0.000, E1   -25.236, E3 -443442.637}
SPL {X  -158.491, Y  +360.654, Z    +0.000, E1   -25.188, E3 -443454.377}
SPL {X  -158.127, Y  +358.155, Z    +0.000, E1   -25.126, E3 -443465.997}
SPL {X  -158.095, Y  +357.947, Z    +0.000, E1   -21.741, E3 -443497.569}
ENDSPLINE

SPLINE
SPL {X  -158.454, Y  +360.384, Z    +0.000, E1   -19.366, E3 -443509.720}
SPL {X  -159.737, Y  +373.507, Z    +0.000, E1   -10.311, E3 -443531.755}
SPL {X  -159.990, Y  +382.574, Z    +0.000, E1    -4.463, E3 -443538.443}
SPL {X  -159.990, Y  +387.496, Z    +0.000, E1    -1.004, E3 -443541.188}
SPL {X  -159.990, Y  +395.121, Z    +0.000, E1    +4.514, E3 -443545.500}
SPL {X  -159.990, Y  +407.941, Z    +0.000, E1   +14.126, E3 -443557.575}
SPL {X  -159.990, Y  +418.671, Z    +0.000, E1   +19.855, E3 -443576.991}
SPL {X  -159.990, Y  +429.878, Z    +0.000, E1   +23.330, E3 -443607.046}
SPL {X  -159.990, Y  +432.766, Z    +0.000, E1   +23.321, E3 -443621.269}
SPL {X  -159.990, Y  +434.794, Z    +0.000, E1   +23.304, E3 -443631.300}
SPL {X  -159.990, Y  +437.007, Z    +0.000, E1   +23.323, E3 -443642.152}
SPL {X  -159.990, Y  +439.778, Z    +0.000, E1   +23.323, E3 -443655.785}
SPL {X  -159.990, Y  +442.945, Z    +0.000, E1   +23.339, E3 -443671.349}
SPL {X  -159.990, Y  +446.037, Z    +0.000, E1   +23.324, E3 -443686.599}
SPL {X  -159.990, Y  +448.797, Z    +0.000, E1   +23.331, E3 -443700.129}
SPL {X  -159.990, Y  +451.747, Z    +0.000, E1   +23.333, E3 -443714.677}
SPL {X  -159.990, Y  +455.185, Z    +0.000, E1   +23.350, E3 -443731.537}
SPL {X  -159.990, Y  +458.265, Z    +0.000, E1   +23.328, E3 -443746.724}
SPL {X  -159.990, Y  +460.492, Z    +0.000, E1   +23.317, E3 -443757.723}
SPL {X  -159.990, Y  +462.929, Z    +0.000, E1   +23.331, E3 -443769.679}
SPL {X  -159.990, Y  +465.027, Z    +0.000, E1   +23.313, E3 -443780.031}
SPL {X  -159.990, Y  +466.881, Z    +0.000, E1   +23.322, E3 -443789.141}
SPL {X  -159.990, Y  +468.951, Z    +0.000, E1   +23.319, E3 -443799.333}
SPL {X  -159.990, Y  +471.818, Z    +0.000, E1   +23.351, E3 -443813.380}
SPL {X  -159.990, Y  +474.801, Z    +0.000, E1   +23.320, E3 -443828.156}
SPL {X  -159.990, Y  +476.830, Z    +0.000, E1   +23.323, E3 -443838.135}
SPL {X  -159.990, Y  +479.553, Z    +0.000, E1   +23.328, E3 -443851.537}
SPL {X  -159.990, Y  +482.950, Z    +0.000, E1   +23.350, E3 -443868.209}
SPL {X  -159.990, Y  +486.109, Z    +0.000, E1   +23.322, E3 -443883.825}
SPL {X  -159.990, Y  +488.481, Z    +0.000, E1   +23.319, E3 -443895.505}
SPL {X  -159.990, Y  +491.454, Z    +0.000, E1   +23.343, E3 -443910.085}
SPL {X  -159.990, Y  +494.937, Z    +0.000, E1   +23.343, E3 -443927.229}
SPL {X  -159.990, Y  +497.668, Z    +0.000, E1   +23.317, E3 -443940.722}
SPL {X  -159.990, Y  +499.995, Z    +0.000, E1   +23.324, E3 -443952.160}
SPL {X  -159.990, Y  +502.456, Z    +0.000, E1   +23.324, E3 -443964.274}
SPL {X  -159.990, Y  +504.508, Z    +0.000, E1   +23.311, E3 -443974.408}
SPL {X  -159.990, Y  +506.420, Z    +0.000, E1   +23.317, E3 -443983.801}
SPL {X  -159.990, Y  +508.862, Z    +0.000, E1   +23.328, E3 -443995.794}
SPL {X  -159.990, Y  +511.771, Z    +0.000, E1   +23.331, E3 -444010.116}
SPL {X  -159.990, Y  +514.016, Z    +0.000, E1   +23.308, E3 -444021.220}
SPL {X  -159.990, Y  +516.860, Z    +0.000, E1   +23.355, E3 -444035.106}
SPL {X  -159.990, Y  +520.719, Z    +0.000, E1   +23.363, E3 -444054.016}
SPL {X  -159.990, Y  +523.968, Z    +0.000, E1   +23.332, E3 -444070.101}
SPL {X  -159.990, Y  +526.466, Z    +0.000, E1   +23.320, E3 -444082.444}
SPL {X  -159.990, Y  +528.815, Z    +0.000, E1   +23.322, E3 -444094.004}
SPL {X  -159.990, Y  +531.246, Z    +0.000, E1   +23.325, E3 -444105.942}
SPL {X  -159.990, Y  +533.354, Z    +0.000, E1   +23.318, E3 -444116.328}
SPL {X  -159.990, Y  +534.931, Z    +0.000, E1   +23.312, E3 -444124.122}
SPL {X  -159.990, Y  +537.024, Z    +0.000, E1   +23.321, E3 -444134.421}
SPL {X  -159.990, Y  +539.129, Z    +0.000, E1   +23.310, E3 -444144.804}
SPL {X  -159.990, Y  +541.183, Z    +0.000, E1   +23.319, E3 -444154.901}
SPL {X  -159.990, Y  +544.314, Z    +0.000, E1   +23.352, E3 -444170.229}
SPL {X  -159.990, Y  +548.126, Z    +0.000, E1   +23.354, E3 -444188.984}
SPL {X  -159.990, Y  +551.344, Z    +0.000, E1   +23.327, E3 -444204.876}
SPL {X  -159.990, Y  +553.642, Z    +0.000, E1   +23.319, E3 -444216.194}
SPL {X  -159.990, Y  +556.481, Z    +0.000, E1   +23.354, E3 -444230.101}
SPL {X  -159.990, Y  +559.475, Z    +0.000, E1   +23.321, E3 -444244.907}
SPL {X  -159.990, Y  +561.830, Z    +0.000, E1   +23.325, E3 -444256.492}
SPL {X  -159.990, Y  +564.273, Z    +0.000, E1   +23.325, E3 -444268.516}
SPL {X  -159.990, Y  +566.342, Z    +0.000, E1   +23.314, E3 -444278.720}
SPL {X  -159.990, Y  +568.184, Z    +0.000, E1   +23.317, E3 -444287.781}
SPL {X  -159.990, Y  +570.560, Z    +0.000, E1   +23.333, E3 -444299.441}
SPL {X  -159.990, Y  +572.975, Z    +0.000, E1   +23.316, E3 -444311.361}
SPL {X  -159.990, Y  +575.097, Z    +0.000, E1   +23.325, E3 -444321.787}
SPL {X  -159.990, Y  +578.356, Z    +0.000, E1   +23.358, E3 -444337.759}
SPL {X  -159.990, Y  +582.292, Z    +0.000, E1   +23.360, E3 -444357.076}
SPL {X  -159.990, Y  +585.165, Z    +0.000, E1   +23.322, E3 -444371.318}
SPL {X  -159.990, Y  +587.388, Z    +0.000, E1   +23.328, E3 -444382.231}
SPL {X  -159.990, Y  +590.594, Z    +0.000, E1   +23.363, E3 -444397.923}
SPL {X  -159.990, Y  +594.301, Z    +0.000, E1   +23.358, E3 -444416.128}
SPL {X  -159.990, Y  +597.981, Z    +0.000, E1   +23.373, E3 -444434.176}
SPL {X  -159.990, Y  +600.935, Z    +0.000, E1   +23.343, E3 -444448.708}
SPL {X  -159.990, Y  +603.047, Z    +0.000, E1   +23.344, E3 -444459.094}
SPL {X  -159.990, Y  +605.187, Z    +0.000, E1   +23.344, E3 -444469.616}
SPL {X  -159.990, Y  +607.319, Z    +0.000, E1   +23.353, E3 -444480.078}
SPL {X  -159.990, Y  +610.569, Z    +0.000, E1   +23.372, E3 -444496.043}
SPL {X  -159.990, Y  +613.591, Z    +0.000, E1   +23.342, E3 -444510.971}
SPL {X  -159.990, Y  +615.604, Z    +0.000, E1   +23.330, E3 -444520.910}
SPL {X  -159.990, Y  +618.445, Z    +0.000, E1   +23.368, E3 -444534.823}
SPL {X  -159.990, Y  +621.517, Z    +0.000, E1   +23.337, E3 -444549.987}
SPL {X  -159.990, Y  +623.764, Z    +0.000, E1   +23.335, E3 -444561.037}
SPL {X  -159.990, Y  +625.941, Z    +0.000, E1   +23.337, E3 -444571.729}
SPL {X  -159.990, Y  +628.611, Z    +0.000, E1   +23.357, E3 -444584.807}
SPL {X  -159.990, Y  +631.169, Z    +0.000, E1   +23.338, E3 -444597.412}
SPL {X  -159.990, Y  +633.318, Z    +0.000, E1   +23.339, E3 -444608.001}
SPL {X  -159.990, Y  +635.650, Z    +0.000, E1   +23.339, E3 -444619.472}
SPL {X  -159.990, Y  +637.839, Z    +0.000, E1   +23.335, E3 -444630.282}
SPL {X  -159.990, Y  +640.072, Z    +0.000, E1   +23.325, E3 -444641.314}
SPL {X  -159.990, Y  +642.230, Z    +0.000, E1   +23.323, E3 -444651.996}
SPL {X  -159.990, Y  +645.287, Z    +0.000, E1   +23.340, E3 -444667.022}
SPL {X  -159.990, Y  +648.792, Z    +0.000, E1   +23.346, E3 -444684.280}
SPL {X  -159.990, Y  +652.623, Z    +0.000, E1   +23.348, E3 -444703.115}
SPL {X  -159.990, Y  +656.380, Z    +0.000, E1   +23.347, E3 -444721.610}
SPL {X  -159.990, Y  +659.180, Z    +0.000, E1   +23.314, E3 -444735.458}
SPL {X  -159.990, Y  +661.392, Z    +0.000, E1   +23.318, E3 -444746.352}
SPL {X  -159.990, Y  +663.662, Z    +0.000, E1   +23.322, E3 -444757.476}
SPL {X  -159.990, Y  +665.964, Z    +0.000, E1   +23.328, E3 -444768.766}
SPL {X  -159.990, Y  +668.989, Z    +0.000, E1   +23.359, E3 -444783.602}
SPL {X  -159.990, Y  +671.893, Z    +0.000, E1   +23.319, E3 -444797.982}
SPL {X  -159.974, Y  +673.789, Z    +0.000, E1   +23.323, E3 -444807.298}
SPL {X  -159.924, Y  +676.110, Z    +0.000, E1   +23.320, E3 -444818.783}
SPL {X  -159.801, Y  +679.265, Z    +0.000, E1   +23.327, E3 -444834.401}
SPL {X  -159.626, Y  +682.287, Z    +0.000, E1   +23.280, E3 -444849.500}
SPL {X  -159.462, Y  +684.486, Z    +0.000, E1   +23.258, E3 -444860.499}
SPL {X  -159.246, Y  +686.911, Z    +0.000, E1   +23.230, E3 -444872.661}
SPL {X  -159.019, Y  +689.098, Z    +0.000, E1   +23.200, E3 -444883.663}
SPL {X  -158.660, Y  +692.086, Z    +0.000, E1   +23.176, E3 -444898.707}
ENDSPLINE

SPLINE
SPL {X  -159.063, Y  +688.696, Z    +0.000, E1   +17.094, E3 -444940.988}
SPL {X  -159.967, Y  +674.206, Z    +0.000, E1    +6.731, E3 -444963.801}
SPL {X  -159.990, Y  +665.270, Z    +0.000, E1    +0.699, E3 -444969.970}
SPL {X  -159.990, Y  +658.009, Z    +0.000, E1    -4.774, E3 -444974.547}
SPL {X  -159.990, Y  +651.567, Z    +0.000, E1    -9.674, E3 -444979.951}
SPL {X  -159.990, Y  +637.762, Z    +0.000, E1   -18.345, E3 -444997.309}
SPL {X  -159.990, Y  +626.382, Z    +0.000, E1   -22.040, E3 -445029.358}
SPL {X  -159.990, Y  +623.760, Z    +0.000, E1   -22.031, E3 -445043.136}
SPL {X  -159.990, Y  +621.334, Z    +0.000, E1   -22.029, E3 -445055.862}
SPL {X  -159.990, Y  +618.387, Z    +0.000, E1   -22.057, E3 -445071.252}
SPL {X  -159.990, Y  +615.830, Z    +0.000, E1   -22.023, E3 -445084.743}
SPL {X  -159.990, Y  +614.007, Z    +0.000, E1   -22.018, E3 -445094.321}
SPL {X  -159.990, Y  +611.459, Z    +0.000, E1   -22.053, E3 -445107.608}
SPL {X  -159.990, Y  +608.810, Z    +0.000, E1   -22.023, E3 -445121.576}
SPL {X  -159.990, Y  +605.804, Z    +0.000, E1   -22.064, E3 -445137.221}
SPL {X  -159.990, Y  +602.819, Z    +0.000, E1   -22.037, E3 -445152.892}
SPL {X  -159.990, Y  +600.642, Z    +0.000, E1   -22.032, E3 -445164.320}
SPL {X  -159.990, Y  +598.568, Z    +0.000, E1   -22.046, E3 -445175.113}
SPL {X  -159.990, Y  +596.440, Z    +0.000, E1   -22.036, E3 -445186.295}
SPL {X  -159.990, Y  +593.768, Z    +0.000, E1   -22.071, E3 -445200.227}
SPL {X  -159.990, Y  +590.068, Z    +0.000, E1   -22.076, E3 -445219.596}
SPL {X  -159.990, Y  +587.130, Z    +0.000, E1   -22.046, E3 -445235.033}
SPL {X  -159.990, Y  +585.120, Z    +0.000, E1   -22.045, E3 -445245.534}
SPL {X  -159.990, Y  +583.118, Z    +0.000, E1   -22.052, E3 -445256.021}
SPL {X  -159.990, Y  +580.862, Z    +0.000, E1   -22.049, E3 -445267.859}
SPL {X  -159.990, Y  +578.386, Z    +0.000, E1   -22.057, E3 -445280.814}
SPL {X  -159.990, Y  +576.252, Z    +0.000, E1   -22.038, E3 -445292.037}
SPL {X  -159.990, Y  +574.280, Z    +0.000, E1   -22.051, E3 -445302.331}
SPL {X  -159.990, Y  +571.711, Z    +0.000, E1   -22.058, E3 -445315.805}
SPL {X  -159.990, Y  +569.285, Z    +0.000, E1   -22.044, E3 -445328.530}
SPL {X  -159.990, Y  +567.211, Z    +0.000, E1   -22.046, E3 -445339.391}
SPL {X  -159.990, Y  +565.039, Z    +0.000, E1   -22.047, E3 -445350.769}
SPL {X  -159.990, Y  +562.755, Z    +0.000, E1   -22.047, E3 -445362.754}
SPL {X  -159.990, Y  +559.661, Z    +0.000, E1   -22.078, E3 -445378.886}
SPL {X  -159.990, Y  +556.672, Z    +0.000, E1   -22.055, E3 -445394.561}
SPL {X  -159.990, Y  +553.726, Z    +0.000, E1   -22.080, E3 -445409.923}
SPL {X  -159.990, Y  +550.886, Z    +0.000, E1   -22.056, E3 -445424.862}
SPL {X  -159.990, Y  +548.814, Z    +0.000, E1   -22.049, E3 -445435.707}
SPL {X  -159.990, Y  +546.122, Z    +0.000, E1   -22.088, E3 -445449.721}
SPL {X  -159.990, Y  +542.390, Z    +0.000, E1   -22.086, E3 -445469.303}
SPL {X  -159.990, Y  +539.341, Z    +0.000, E1   -22.056, E3 -445485.324}
SPL {X  -159.990, Y  +536.301, Z    +0.000, E1   -22.084, E3 -445501.179}
SPL {X  -159.990, Y  +533.389, Z    +0.000, E1   -22.057, E3 -445516.486}
SPL {X  -159.990, Y  +531.347, Z    +0.000, E1   -22.052, E3 -445527.187}
SPL {X  -159.990, Y  +529.626, Z    +0.000, E1   -22.051, E3 -445536.184}
SPL {X  -159.990, Y  +527.412, Z    +0.000, E1   -22.067, E3 -445547.737}
SPL {X  -159.990, Y  +524.425, Z    +0.000, E1   -22.078, E3 -445563.369}
SPL {X  -159.990, Y  +521.599, Z    +0.000, E1   -22.060, E3 -445578.211}
SPL {X  -159.990, Y  +519.209, Z    +0.000, E1   -22.063, E3 -445590.686}
SPL {X  -159.990, Y  +516.651, Z    +0.000, E1   -22.071, E3 -445604.066}
SPL {X  -159.990, Y  +514.122, Z    +0.000, E1   -22.061, E3 -445617.338}
SPL {X  -159.990, Y  +511.670, Z    +0.000, E1   -22.064, E3 -445630.188}
SPL {X  -159.990, Y  +506.947, Z    +0.000, E1   -23.726, E3 -445640.216}
SPL {X  -159.990, Y  +496.921, Z    +0.000, E1   -28.340, E3 -445648.965}
SPL {X  -159.990, Y  +495.822, Z    +0.000, E1   -27.449, E3 -445659.713}
SPL {X  -159.990, Y  +494.952, Z    +0.000, E1   -26.628, E3 -445669.296}
SPL {X  -159.990, Y  +493.896, Z    +0.000, E1   -25.736, E3 -445680.626}
SPL {X  -159.990, Y  +491.647, Z    +0.000, E1   -25.401, E3 -445693.161}
SPL {X  -159.990, Y  +488.807, Z    +0.000, E1   -25.397, E3 -445705.860}
SPL {X  -159.990, Y  +486.070, Z    +0.000, E1   -25.399, E3 -445718.091}
SPL {X  -159.990, Y  +482.821, Z    +0.000, E1   -25.411, E3 -445732.592}
SPL {X  -159.990, Y  +480.183, Z    +0.000, E1   -25.384, E3 -445744.432}
SPL {X  -159.990, Y  +478.407, Z    +0.000, E1   -25.384, E3 -445752.373}
SPL {X  -159.990, Y  +475.940, Z    +0.000, E1   -25.403, E3 -445763.363}
SPL {X  -159.990, Y  +473.026, Z    +0.000, E1   -25.399, E3 -445776.393}
SPL {X  -159.990, Y  +470.047, Z    +0.000, E1   -25.402, E3 -445789.711}
SPL {X  -159.990, Y  +467.082, Z    +0.000, E1   -25.399, E3 -445802.958}
SPL {X  -159.990, Y  +464.919, Z    +0.000, E1   -25.381, E3 -445812.685}
SPL {X  -159.990, Y  +462.520, Z    +0.000, E1   -25.400, E3 -445823.359}
SPL {X  -159.990, Y  +460.081, Z    +0.000, E1   -25.390, E3 -445834.261}
SPL {X  -159.990, Y  +457.497, Z    +0.000, E1   -25.403, E3 -445845.785}
SPL {X  -159.990, Y  +454.323, Z    +0.000, E1   -25.412, E3 -445859.944}
SPL {X  -159.990, Y  +451.400, Z    +0.000, E1   -25.397, E3 -445873.035}
SPL {X  -159.990, Y  +448.503, Z    +0.000, E1   -25.410, E3 -445885.953}
SPL {X  -159.990, Y  +445.108, Z    +0.000, E1   -25.407, E3 -445901.191}
SPL {X  -159.990, Y  +441.797, Z    +0.000, E1   -25.390, E3 -445916.070}
SPL {X  -159.990, Y  +439.442, Z    +0.000, E1   -25.369, E3 -445926.647}
SPL {X  -159.990, Y  +436.316, Z    +0.000, E1   -25.420, E3 -445940.529}
SPL {X  -159.990, Y  +432.613, Z    +0.000, E1   -25.390, E3 -445957.154}
SPL {X  -159.990, Y  +429.079, Z    +0.000, E1   -25.407, E3 -445972.925}
SPL {X  -159.990, Y  +426.149, Z    +0.000, E1   -25.374, E3 -445986.087}
SPL {X  -159.990, Y  +423.417, Z    +0.000, E1   -25.400, E3 -445998.252}
SPL {X  -159.990, Y  +420.283, Z    +0.000, E1   -25.386, E3 -446012.297}
SPL {X  -159.990, Y  +417.514, Z    +0.000, E1   -25.386, E3 -446024.681}
SPL {X  -159.990, Y  +414.805, Z    +0.000, E1   -25.385, E3 -446036.801}
SPL {X  -159.990, Y  +411.282, Z    +0.000, E1   -25.413, E3 -446052.502}
SPL {X  -159.990, Y  +408.351, Z    +0.000, E1   -25.372, E3 -446065.689}
SPL {X  -159.990, Y  +405.773, Z    +0.000, E1   -25.398, E3 -446077.142}
SPL {X  -159.990, Y  +402.805, Z    +0.000, E1   -25.389, E3 -446090.428}
SPL {X  -159.990, Y  +400.083, Z    +0.000, E1   -25.388, E3 -446102.604}
SPL {X  -159.990, Y  +396.740, Z    +0.000, E1   -25.410, E3 -446117.529}
SPL {X  -159.990, Y  +392.622, Z    +0.000, E1   -25.413, E3 -446135.957}
SPL {X  -159.990, Y  +388.328, Z    +0.000, E1   -25.413, E3 -446155.185}
SPL {X  -159.990, Y  +384.900, Z    +0.000, E1   -25.383, E3 -446170.547}
SPL {X  -159.990, Y  +382.110, Z    +0.000, E1   -25.393, E3 -446182.993}
SPL {X  -159.961, Y  +379.439, Z    +0.000, E1   -25.380, E3 -446194.973}
SPL {X  -159.894, Y  +376.959, Z    +0.000, E1   -25.370, E3 -446206.150}
SPL {X  -159.784, Y  +374.382, Z    +0.000, E1   -25.356, E3 -446217.791}
SPL {X  -159.621, Y  +371.640, Z    +0.000, E1   -25.335, E3 -446230.231}
SPL {X  -159.406, Y  +368.844, Z    +0.000, E1   -25.307, E3 -446242.944}
SPL {X  -159.144, Y  +366.072, Z    +0.000, E1   -25.281, E3 -446255.551}
SPL {X  -158.822, Y  +363.200, Z    +0.000, E1   -25.236, E3 -446268.724}
SPL {X  -158.491, Y  +360.654, Z    +0.000, E1   -25.188, E3 -446280.464}
SPL {X  -158.127, Y  +358.155, Z    +0.000, E1   -25.126, E3 -446292.084}
SPL {X  -158.095, Y  +357.947, Z    +0.000, E1   -21.741, E3 -446323.656}
ENDSPLINE

SPLINE
SPL {X  -158.454, Y  +360.384, Z    +0.000, E1   -19.366, E3 -446335.807}
SPL {X  -159.737, Y  +373.507, Z    +0.000, E1   -10.311, E3 -446357.842}
SPL {X  -159.990, Y  +382.574, Z    +0.000, E1    -4.463, E3 -446364.530}
SPL {X  -159.990, Y  +389.909, Z    +0.000, E1    +0.662, E3 -446368.545}
SPL {X  -159.990, Y  +396.289, Z    +0.000, E1    +5.500, E3 -446372.325}
SPL {X  -159.990, Y  +407.941, Z    +0.000, E1   +14.126, E3 -446383.662}
SPL {X  -159.990, Y  +418.671, Z    +0.000, E1   +19.855, E3 -446403.078}
SPL {X  -159.990, Y  +428.534, Z    +0.000, E1   +23.299, E3 -446426.598}
SPL {X  -159.990, Y  +430.313, Z    +0.000, E1   +23.313, E3 -446435.311}
SPL {X  -159.990, Y  +432.766, Z    +0.000, E1   +23.321, E3 -446447.356}
SPL {X  -159.990, Y  +434.794, Z    +0.000, E1   +23.304, E3 -446457.387}
SPL {X  -159.990, Y  +437.007, Z    +0.000, E1   +23.323, E3 -446468.239}
SPL {X  -159.990, Y  +439.778, Z    +0.000, E1   +23.323, E3 -446481.872}
SPL {X  -159.990, Y  +442.010, Z    +0.000, E1   +23.308, E3 -446492.893}
SPL {X  -159.990, Y  +443.729, Z    +0.000, E1   +23.310, E3 -446501.349}
SPL {X  -159.990, Y  +446.037, Z    +0.000, E1   +23.324, E3 -446512.686}
SPL {X  -159.990, Y  +449.434, Z    +0.000, E1   +23.356, E3 -446529.307}
SPL {X  -159.990, Y  +453.256, Z    +0.000, E1   +23.349, E3 -446548.142}
SPL {X  -159.990, Y  +455.953, Z    +0.000, E1   +23.320, E3 -446561.456}
SPL {X  -159.990, Y  +458.265, Z    +0.000, E1   +23.328, E3 -446572.811}
SPL {X  -159.990, Y  +461.258, Z    +0.000, E1   +23.344, E3 -446587.527}
SPL {X  -159.990, Y  +464.382, Z    +0.000, E1   +23.332, E3 -446602.908}
SPL {X  -159.990, Y  +466.881, Z    +0.000, E1   +23.322, E3 -446615.228}
SPL {X  -159.990, Y  +468.951, Z    +0.000, E1   +23.319, E3 -446625.420}
SPL {X  -159.990, Y  +470.991, Z    +0.000, E1   +23.322, E3 -446635.450}
SPL {X  -159.990, Y  +474.027, Z    +0.000, E1   +23.352, E3 -446650.354}
SPL {X  -159.990, Y  +477.600, Z    +0.000, E1   +23.351, E3 -446667.957}
SPL {X  -159.990, Y  +481.169, Z    +0.000, E1   +23.337, E3 -446685.555}
SPL {X  -159.990, Y  +483.782, Z    +0.000, E1   +23.316, E3 -446698.459}
SPL {X  -159.990, Y  +486.109, Z    +0.000, E1   +23.322, E3 -446709.912}
SPL {X  -159.990, Y  +489.247, Z    +0.000, E1   +23.348, E3 -446725.299}
SPL {X  -159.990, Y  +493.031, Z    +0.000, E1   +23.350, E3 -446743.923}
SPL {X  -159.990, Y  +496.869, Z    +0.000, E1   +23.349, E3 -446762.814}
SPL {X  -159.990, Y  +499.995, Z    +0.000, E1   +23.324, E3 -446778.247}
SPL {X  -159.990, Y  +502.456, Z    +0.000, E1   +23.324, E3 -446790.361}
SPL {X  -159.990, Y  +505.646, Z    +0.000, E1   +23.350, E3 -446806.017}
SPL {X  -159.990, Y  +508.862, Z    +0.000, E1   +23.328, E3 -446821.881}
SPL {X  -159.990, Y  +510.971, Z    +0.000, E1   +23.308, E3 -446832.309}
SPL {X  -159.990, Y  +513.289, Z    +0.000, E1   +23.332, E3 -446843.675}
SPL {X  -159.990, Y  +516.860, Z    +0.000, E1   +23.355, E3 -446861.193}
SPL {X  -159.990, Y  +520.719, Z    +0.000, E1   +23.363, E3 -446880.103}
SPL {X  -159.990, Y  +523.968, Z    +0.000, E1   +23.332, E3 -446896.188}
SPL {X  -159.990, Y  +526.466, Z    +0.000, E1   +23.320, E3 -446908.531}
SPL {X  -159.990, Y  +528.815, Z    +0.000, E1   +23.322, E3 -446920.091}
SPL {X  -159.990, Y  +531.246, Z    +0.000, E1   +23.325, E3 -446932.029}
SPL {X  -159.990, Y  +533.354, Z    +0.000, E1   +23.318, E3 -446942.415}
SPL {X  -159.990, Y  +534.931, Z    +0.000, E1   +23.312, E3 -446950.209}
SPL {X  -159.990, Y  +537.024, Z    +0.000, E1   +23.321, E3 -446960.508}
SPL {X  -159.990, Y  +539.129, Z    +0.000, E1   +23.310, E3 -446970.891}
SPL {X  -159.990, Y  +541.183, Z    +0.000, E1   +23.319, E3 -446980.987}
SPL {X  -159.990, Y  +544.314, Z    +0.000, E1   +23.352, E3 -446996.316}
SPL {X  -159.990, Y  +548.126, Z    +0.000, E1   +23.354, E3 -447015.071}
SPL {X  -159.990, Y  +551.344, Z    +0.000, E1   +23.327, E3 -447030.963}
SPL {X  -159.990, Y  +553.642, Z    +0.000, E1   +23.319, E3 -447042.281}
SPL {X  -159.990, Y  +556.481, Z    +0.000, E1   +23.354, E3 -447056.188}
SPL {X  -159.990, Y  +559.475, Z    +0.000, E1   +23.321, E3 -447070.994}
SPL {X  -159.990, Y  +561.830, Z    +0.000, E1   +23.325, E3 -447082.579}
SPL {X  -159.990, Y  +564.273, Z    +0.000, E1   +23.325, E3 -447094.603}
SPL {X  -159.990, Y  +567.351, Z    +0.000, E1   +23.348, E3 -447109.699}
SPL {X  -159.990, Y  +570.560, Z    +0.000, E1   +23.333, E3 -447125.528}
SPL {X  -159.990, Y  +572.975, Z    +0.000, E1   +23.316, E3 -447137.448}
SPL {X  -159.990, Y  +575.097, Z    +0.000, E1   +23.325, E3 -447147.874}
SPL {X  -159.990, Y  +577.540, Z    +0.000, E1   +23.325, E3 -447159.903}
SPL {X  -159.990, Y  +580.312, Z    +0.000, E1   +23.340, E3 -447173.485}
SPL {X  -159.990, Y  +583.018, Z    +0.000, E1   +23.331, E3 -447186.790}
SPL {X  -159.990, Y  +585.165, Z    +0.000, E1   +23.322, E3 -447197.405}
SPL {X  -159.990, Y  +587.388, Z    +0.000, E1   +23.328, E3 -447208.318}
SPL {X  -159.990, Y  +590.594, Z    +0.000, E1   +23.363, E3 -447224.010}
SPL {X  -159.990, Y  +593.168, Z    +0.000, E1   +23.322, E3 -447236.722}
SPL {X  -159.990, Y  +595.589, Z    +0.000, E1   +23.356, E3 -447248.559}
SPL {X  -159.990, Y  +598.571, Z    +0.000, E1   +23.347, E3 -447263.202}
SPL {X  -159.990, Y  +600.935, Z    +0.000, E1   +23.343, E3 -447274.795}
SPL {X  -159.990, Y  +603.047, Z    +0.000, E1   +23.344, E3 -447285.181}
SPL {X  -159.990, Y  +605.187, Z    +0.000, E1   +23.344, E3 -447295.703}
SPL {X  -159.990, Y  +607.319, Z    +0.000, E1   +23.353, E3 -447306.165}
SPL {X  -159.990, Y  +609.514, Z    +0.000, E1   +23.337, E3 -447316.994}
SPL {X  -159.990, Y  +611.376, Z    +0.000, E1   +23.336, E3 -447326.181}
SPL {X  -159.990, Y  +613.591, Z    +0.000, E1   +23.342, E3 -447337.058}
SPL {X  -159.990, Y  +615.604, Z    +0.000, E1   +23.330, E3 -447346.996}
SPL {X  -159.990, Y  +617.623, Z    +0.000, E1   +23.337, E3 -447356.927}
SPL {X  -159.990, Y  +620.788, Z    +0.000, E1   +23.368, E3 -447372.432}
SPL {X  -159.990, Y  +623.764, Z    +0.000, E1   +23.335, E3 -447387.124}
SPL {X  -159.990, Y  +625.941, Z    +0.000, E1   +23.337, E3 -447397.816}
SPL {X  -159.990, Y  +628.611, Z    +0.000, E1   +23.357, E3 -447410.894}
SPL {X  -159.990, Y  +631.169, Z    +0.000, E1   +23.338, E3 -447423.499}
SPL {X  -159.990, Y  +633.318, Z    +0.000, E1   +23.339, E3 -447434.088}
SPL {X  -159.990, Y  +635.650, Z    +0.000, E1   +23.339, E3 -447445.559}
SPL {X  -159.990, Y  +637.839, Z    +0.000, E1   +23.335, E3 -447456.369}
SPL {X  -159.990, Y  +640.072, Z    +0.000, E1   +23.325, E3 -447467.401}
SPL {X  -159.990, Y  +642.230, Z    +0.000, E1   +23.323, E3 -447478.083}
SPL {X  -159.990, Y  +645.287, Z    +0.000, E1   +23.340, E3 -447493.109}
SPL {X  -159.990, Y  +648.792, Z    +0.000, E1   +23.346, E3 -447510.367}
SPL {X  -159.990, Y  +652.623, Z    +0.000, E1   +23.348, E3 -447529.202}
SPL {X  -159.990, Y  +656.380, Z    +0.000, E1   +23.347, E3 -447547.697}
SPL {X  -159.990, Y  +659.180, Z    +0.000, E1   +23.314, E3 -447561.545}
SPL {X  -159.990, Y  +661.392, Z    +0.000, E1   +23.318, E3 -447572.439}
SPL {X  -159.990, Y  +663.662, Z    +0.000, E1   +23.322, E3 -447583.563}
SPL {X  -159.990, Y  +665.964, Z    +0.000, E1   +23.328, E3 -447594.853}
SPL {X  -159.990, Y  +668.989, Z    +0.000, E1   +23.359, E3 -447609.689}
SPL {X  -159.983, Y  +672.946, Z    +0.000, E1   +23.359, E3 -447629.170}
SPL {X  -159.924, Y  +676.110, Z    +0.000, E1   +23.320, E3 -447644.870}
SPL {X  -159.801, Y  +679.265, Z    +0.000, E1   +23.327, E3 -447660.488}
SPL {X  -159.626, Y  +682.287, Z    +0.000, E1   +23.280, E3 -447675.587}
SPL {X  -159.462, Y  +684.486, Z    +0.000, E1   +23.258, E3 -447686.586}
SPL {X  -159.246, Y  +686.911, Z    +0.000, E1   +23.230, E3 -447698.748}
SPL {X  -159.019, Y  +689.098, Z    +0.000, E1   +23.200, E3 -447709.750}
SPL {X  -158.660, Y  +692.086, Z    +0.000, E1   +23.176, E3 -447724.794}
ENDSPLINE

